KUKA KRL program: MyProgram_136().src

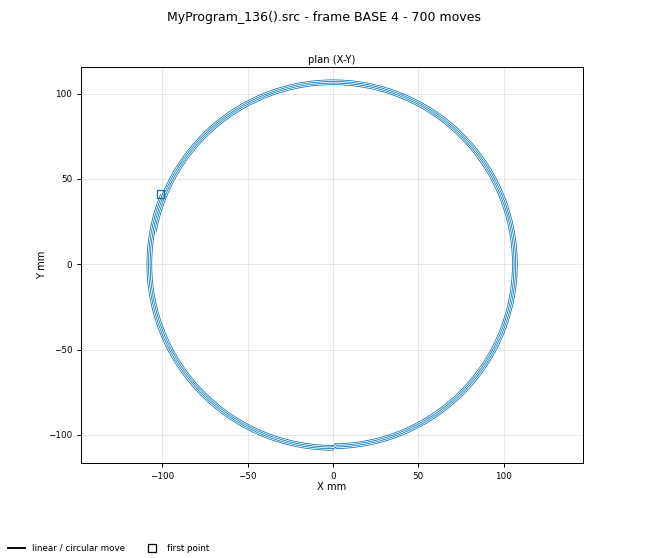
[picture p0: tool path of MyProgram_136().src in frame BASE 4, 700 of 700 moves have a stored position in this frame; points joined in program order, loops and branches not executed]
&ACCESS RVP
&REL 1
&PARAM TEMPLATE = C:\KRC\Roboter\Template\vorgabe
&PARAM EDITMASK = *
DEF MyProgram_136()
; ---- Setting reference (Base) ----
$BASE = BASE_DATA[4]

; --------------------------
; ---- Setting tool (TCP) ----
$TOOL = TOOL_DATA[3]
; --------------------------

$VEL.CP = VEL_APROX_PRINT
Startdeposition()
$VEL.CP = VEL_PRINT
LIN {X -101.0459,Y 40.9504,Z 110,A 153.8503,B 24.9356,C -1.8541,E1 24.8512,E2 291.8674} C_DIS
LIN {X -102.4048,Y 37.4224,Z 110,A 155.9368,B 24.9357,C -1.8516,E1 24.8492,E2 289.7749} C_DIS
LIN {X -103.4357,Y 34.473,Z 110,A 157.5676,B 24.9361,C -1.8461,E1 24.8477,E2 288.1481} C_DIS
LIN {X -104.6474,Y 30.5989,Z 110,A 159.7018,B 24.9366,C -1.8394,E1 24.846,E2 286.0176} C_DIS
LIN {X -105.5429,Y 27.3483,Z 110,A 161.5611,B 24.9367,C -1.837,E1 24.8446,E2 284.1531} C_DIS
LIN {X -106.3392,Y 24.0704,Z 110,A 163.3808,B 24.937,C -1.8331,E1 24.8435,E2 282.332} C_DIS
LIN {X -106.8901,Y 21.4916,Z 110,A 164.9562,B 24.9368,C -1.8358,E1 24.8426,E2 280.7408} C_DIS
LIN {X -107.8686,Y 15.8696,Z 110,A 167.7801,B 24.9379,C -1.8195,E1 24.8413,E2 277.9391} C_DIS
LIN {X -108.3438,Y 12.2078,Z 110,A 170.4812,B 24.9364,C -1.8421,E1 24.8404,E2 275.168} C_DIS
LIN {X -108.7748,Y 7.4321,Z 110,A 172.0604,B 24.9394,C -1.7983,E1 24.8401,E2 273.6837} C_DIS
LIN {X -109.0243,Y 1.0365,Z 110,A 175.4778,B 24.94,C -1.7893,E1 24.8398,E2 270.2672} C_DIS
LIN {X -108.9337,Y -4.5435,Z 110,A 179.2186,B 24.9386,C -1.8105,E1 24.8401,E2 266.4534} C_DIS
LIN {X -108.6738,Y -8.7861,Z 110,A -179.1678,B 24.9406,C -1.7797,E1 24.8404,E2 264.9035} C_DIS
LIN {X -108.4394,Y -11.3169,Z 110,A -177.6162,B 24.9404,C -1.7836,E1 24.8409,E2 263.3332} C_DIS
LIN {X -107.6634,Y -17.2072,Z 110,A -174.7453,B 24.9417,C -1.7642,E1 24.842,E2 260.4916} C_DIS
LIN {X -106.9005,Y -21.4409,Z 110,A -172.3194,B 24.9417,C -1.7633,E1 24.8432,E2 258.0534} C_DIS
LIN {X -106.0833,Y -25.1782,Z 110,A -170.3045,B 24.9421,C -1.7572,E1 24.8445,E2 256.0412} C_DIS
LIN {X -105.2578,Y -28.4248,Z 110,A -168.6511,B 24.9427,C -1.7478,E1 24.8456,E2 254.4007} C_DIS
LIN {X -104.3481,Y -31.6078,Z 110,A -166.7945,B 24.9428,C -1.7469,E1 24.8471,E2 252.5355} C_DIS
LIN {X -103.3127,Y -34.8378,Z 110,A -165.0254,B 24.9432,C -1.7411,E1 24.8487,E2 250.7702} C_DIS
LIN {X -102.0795,Y -38.3024,Z 110,A -163.1309,B 24.9437,C -1.7339,E1 24.8505,E2 248.8821} C_DIS
LIN {X -100.0319,Y -43.3688,Z 110,A -160.4375,B 24.9446,C -1.7187,E1 24.8533,E2 246.2098} C_DIS
LIN {X -98.1863,Y -47.399,Z 110,A -157.8891,B 24.9446,C -1.7204,E1 24.8563,E2 243.6435} C_DIS
LIN {X -96.4981,Y -50.7474,Z 110,A -155.8502,B 24.9447,C -1.7176,E1 24.8589,E2 241.6005} C_DIS
LIN {X -94.7103,Y -54.0117,Z 110,A -153.865,B 24.945,C -1.7134,E1 24.8616,E2 239.6149} C_DIS
LIN {X -91.6565,Y -59.0449,Z 110,A -150.4776,B 24.9448,C -1.7165,E1 24.8667,E2 236.2027} C_DIS
LIN {X -88.8476,Y -63.1926,Z 110,A -148.2791,B 24.9463,C -1.6931,E1 24.8701,E2 234.0492} C_DIS
LIN {X -86.6848,Y -66.1302,Z 110,A -146.1765,B 24.9461,C -1.6955,E1 24.8736,E2 231.9307} C_DIS
LIN {X -84.5749,Y -68.8062,Z 110,A -144.3868,B 24.9464,C -1.6912,E1 24.8768,E2 230.1428} C_DIS
LIN {X -82.6969,Y -71.0536,Z 110,A -142.3954,B 24.9455,C -1.7053,E1 24.8805,E2 228.1088} C_DIS
LIN {X -80.2724,Y -73.7802,Z 110,A -140.9176,B 24.9469,C -1.6838,E1 24.8832,E2 226.6757} C_DIS
LIN {X -77.6379,Y -76.5476,Z 110,A -139.1883,B 24.9478,C -1.6686,E1 24.8865,E2 224.9752} C_DIS
LIN {X -75.502,Y -78.6554,Z 110,A -137.3296,B 24.9473,C -1.6763,E1 24.8902,E2 223.0904} C_DIS
LIN {X -72.5889,Y -81.3515,Z 110,A -135.2119,B 24.9475,C -1.6733,E1 24.8946,E2 220.9713} C_DIS
LIN {X -69.8379,Y -83.725,Z 110,A -132.8251,B 24.9466,C -1.6885,E1 24.8998,E2 218.539} C_DIS
LIN {X -66.8378,Y -86.1396,Z 110,A -131.2769,B 24.948,C -1.666,E1 24.9031,E2 217.0388} C_DIS
LIN {X -63.7429,Y -88.455,Z 110,A -129.2893,B 24.9483,C -1.6607,E1 24.9076,E2 215.0566} C_DIS
LIN {X -60.5392,Y -90.6784,Z 110,A -127.116,B 24.9483,C -1.6623,E1 24.9126,E2 212.8724} C_DIS
LIN {X -55.2575,Y -93.9885,Z 110,A -123.6526,B 24.9481,C -1.6649,E1 24.9209,E2 209.392} C_DIS
LIN {X -51.1504,Y -96.2858,Z 110,A -121.304,B 24.9486,C -1.6566,E1 24.9266,E2 207.0566} C_DIS
LIN {X -46.668,Y -98.5376,Z 110,A -118.6742,B 24.9488,C -1.6531,E1 24.9332,E2 204.4282} C_DIS
LIN {X -43.398,Y -100.0191,Z 110,A -116.9327,B 24.9493,C -1.6452,E1 24.9376,E2 202.7013} C_DIS
LIN {X -39.7895,Y -101.5085,Z 110,A -114.827,B 24.9493,C -1.6453,E1 24.9431,E2 200.5906} C_DIS
LIN {X -36.1315,Y -102.8674,Z 110,A -112.8041,B 24.9495,C -1.6424,E1 24.9484,E2 198.5706} C_DIS
LIN {X -33.5707,Y -103.7313,Z 110,A -111.2544,B 24.9492,C -1.6465,E1 24.9525,E2 197.0083} C_DIS
LIN {X -28.2847,Y -105.2957,Z 110,A -108.424,B 24.9495,C -1.6418,E1 24.9601,E2 194.1844} C_DIS
LIN {X -25.199,Y -106.0784,Z 110,A -106.2515,B 24.9483,C -1.6615,E1 24.9662,E2 191.9624} C_DIS
LIN {X -21.329,Y -106.9234,Z 110,A -104.7514,B 24.9498,C -1.6366,E1 24.9701,E2 190.5195} C_DIS
LIN {X -17.6406,Y -107.5923,Z 110,A -102.8021,B 24.9499,C -1.6351,E1 24.9755,E2 188.5718} C_DIS
LIN {X -14.2432,Y -108.0942,Z 110,A -101.1009,B 24.9502,C -1.6305,E1 24.9801,E2 186.8803} C_DIS
LIN {X -11.5445,Y -108.4156,Z 110,A -99.5635,B 24.9499,C -1.6348,E1 24.9844,E2 185.3317} C_DIS
LIN {X -8.3441,Y -108.7091,Z 110,A -97.7326,B 24.9496,C -1.6406,E1 24.9896,E2 183.4862} C_DIS
LIN {X -4.4559,Y -108.9375,Z 110,A -95.6989,B 24.9496,C -1.6402,E1 24.9952,E2 181.4529} C_DIS
LIN {X -0.5852,Y -109.0268,Z 110,A -93.7792,B 24.9499,C -1.6358,E1 25.0006,E2 179.5435} C_DIS
LIN {X -0.5852,Y -109.0268,Z 110,A -93.7792,B 24.9499,C -1.6358,E1 25.0006,E2 179.5435} C_DIS
Enddeposition()
LIN {X 0.7508,Y -108.0795,Z 110,A -93.2455,B 24.9493,C -1.6454,E1 25.0021,E2 178.9871} C_DIS
Startdeposition()
$VEL.CP = VEL_PRINT
LIN {X -2.9231,Y -108.0454,Z 110,A -95.8982,B 24.9511,C -1.6161,E1 24.9945,E2 181.7093} C_DIS
LIN {X -6.8398,Y -107.8686,Z 110,A -97.972,B 24.9511,C -1.6161,E1 24.9888,E2 183.7836} C_DIS
LIN {X -10.1831,Y -107.6038,Z 110,A -99.6434,B 24.9508,C -1.6206,E1 24.9841,E2 185.4454} C_DIS
LIN {X -13.0586,Y -107.2936,Z 110,A -101.1347,B 24.9507,C -1.6224,E1 24.98,E2 186.9331} C_DIS
LIN {X -16.4613,Y -106.8234,Z 110,A -103.3915,B 24.9517,C -1.6054,E1 24.9737,E2 189.2322} C_DIS
LIN {X -19.6265,Y -106.2886,Z 110,A -104.6024,B 24.9505,C -1.6256,E1 24.9705,E2 190.3964} C_DIS
LIN {X -24.2676,Y -105.3247,Z 110,A -107.2289,B 24.9507,C -1.6222,E1 24.9633,E2 193.0342} C_DIS
LIN {X -30.7493,Y -103.618,Z 110,A -110.7194,B 24.9504,C -1.6269,E1 24.9539,E2 196.5189} C_DIS
LIN {X -33.1251,Y -102.8832,Z 110,A -112.13,B 24.9506,C -1.6242,E1 24.9501,E2 197.9384} C_DIS
LIN {X -36.5679,Y -101.7116,Z 110,A -114.1221,B 24.9506,C -1.6233,E1 24.9448,E2 199.9365} C_DIS
LIN {X -39.7247,Y -100.5197,Z 110,A -115.8285,B 24.9503,C -1.6283,E1 24.9404,E2 201.6347} C_DIS
LIN {X -42.6112,Y -99.3323,Z 110,A -117.5613,B 24.9504,C -1.6269,E1 24.9359,E2 203.3748} C_DIS
LIN {X -46.4464,Y -97.5966,Z 110,A -119.5451,B 24.9497,C -1.6392,E1 24.9309,E2 205.3343} C_DIS
LIN {X -48.7324,Y -96.476,Z 110,A -121.188,B 24.9503,C -1.6294,E1 24.9268,E2 207.0049} C_DIS
LIN {X -51.8131,Y -94.8562,Z 110,A -122.9938,B 24.95,C -1.6334,E1 24.9223,E2 208.8063} C_DIS
LIN {X -57.8107,Y -91.3266,Z 110,A -126.8101,B 24.95,C -1.6338,E1 24.9132,E2 212.6331} C_DIS
LIN {X -62.0089,Y -88.5283,Z 110,A -129.597,B 24.95,C -1.6339,E1 24.9067,E2 215.4292} C_DIS
LIN {X -64.932,Y -86.4062,Z 110,A -131.2208,B 24.9491,C -1.6484,E1 24.9031,E2 217.0242} C_DIS
LIN {X -70.239,Y -82.1506,Z 110,A -134.64,B 24.9482,C -1.6623,E1 24.8958,E2 220.4233} C_DIS
LIN {X -72.1623,Y -80.4663,Z 110,A -136.274,B 24.9487,C -1.6543,E1 24.8923,E2 222.0828} C_DIS
LIN {X -75.7805,Y -77.0687,Z 110,A -138.8814,B 24.9483,C -1.6606,E1 24.887,E2 224.6858} C_DIS
LIN {X -78.0174,Y -74.8036,Z 110,A -140.6814,B 24.9483,C -1.66,E1 24.8835,E2 226.4951} C_DIS
LIN {X -82.8135,Y -69.4577,Z 110,A -144.2462,B 24.9472,C -1.6778,E1 24.877,E2 230.0334} C_DIS
LIN {X -86.9571,Y -64.1939,Z 110,A -148.0447,B 24.9472,C -1.6771,E1 24.8704,E2 233.8517} C_DIS
LIN {X -89.1258,Y -61.1493,Z 110,A -150.2115,B 24.9474,C -1.6751,E1 24.8669,E2 236.0338} C_DIS
LIN {X -91.2432,Y -57.941,Z 110,A -152.5341,B 24.9477,C -1.6699,E1 24.8634,E2 238.3808} C_DIS
LIN {X -93.173,Y -54.782,Z 110,A -154.0573,B 24.9464,C -1.6914,E1 24.8613,E2 239.8604} C_DIS
LIN {X -95.078,Y -51.4044,Z 110,A -156.0328,B 24.9458,C -1.7,E1 24.8586,E2 241.8258} C_DIS
LIN {X -96.7287,Y -48.2268,Z 110,A -158.0219,B 24.9458,C -1.7019,E1 24.8561,E2 243.821} C_DIS
LIN {X -98.8506,Y -43.716,Z 110,A -160.6588,B 24.9452,C -1.7096,E1 24.853,E2 246.454} C_DIS
LIN {X -100.8213,Y -38.9567,Z 110,A -163.2646,B 24.9444,C -1.7222,E1 24.8503,E2 249.0443} C_DIS
LIN {X -102.0825,Y -35.517,Z 110,A -165.4232,B 24.9446,C -1.72,E1 24.8483,E2 251.2204} C_DIS
LIN {X -103.0681,Y -32.5499,Z 110,A -167.1107,B 24.9443,C -1.7239,E1 24.8468,E2 252.9084} C_DIS
LIN {X -104.0473,Y -29.2647,Z 110,A -168.7742,B 24.9436,C -1.7351,E1 24.8455,E2 254.5548} C_DIS
LIN {X -104.9195,Y -25.9661,Z 110,A -170.6629,B 24.9434,C -1.7377,E1 24.8442,E2 256.4482} C_DIS
LIN {X -105.7058,Y -22.5552,Z 110,A -172.6177,B 24.9433,C -1.7398,E1 24.843,E2 258.4095} C_DIS
LIN {X -106.6749,Y -17.4029,Z 110,A -175.1438,B 24.9421,C -1.7579,E1 24.8418,E2 260.9075} C_DIS
LIN {X -107.4911,Y -11.3081,Z 110,A -178.2308,B 24.941,C -1.7746,E1 24.8407,E2 263.9731} C_DIS
LIN {X -107.9447,Y -5.5101,Z 110,A 177.6041,B 24.9429,C -1.7449,E1 24.8399,E2 268.2341} C_DIS
LIN {X -108.0802,Y -1.0392,Z 110,A 176.1681,B 24.9402,C -1.7866,E1 24.8399,E2 269.5792} C_DIS
LIN {X -107.8861,Y 6.5706,Z 110,A 170.7512,B 24.9426,C -1.7495,E1 24.8404,E2 275.1172} C_DIS
LIN {X -107.3472,Y 12.601,Z 110,A 169.0253,B 24.9383,C -1.8138,E1 24.8409,E2 276.7001} C_DIS
LIN {X -106.5725,Y 18.0154,Z 110,A 165.5521,B 24.9391,C -1.8021,E1 24.8423,E2 280.222} C_DIS
LIN {X -105.91,Y 21.5708,Z 110,A 163.7053,B 24.9385,C -1.8108,E1 24.8433,E2 282.0589} C_DIS
LIN {X -105.0583,Y 25.3971,Z 110,A 161.6175,B 24.9381,C -1.8171,E1 24.8446,E2 284.1439} C_DIS
LIN {X -104.148,Y 28.9093,Z 110,A 159.1474,B 24.9391,C -1.8033,E1 24.8465,E2 286.6614} C_DIS
LIN {X -103.0003,Y 32.7633,Z 110,A 157.4686,B 24.9375,C -1.8264,E1 24.8478,E2 288.2945} C_DIS
LIN {X -101.7936,Y 36.3402,Z 110,A 155.2258,B 24.9376,C -1.8239,E1 24.8499,E2 290.5562} C_DIS
LIN {X -100.0581,Y 40.873,Z 110,A 152.9865,B 24.9363,C -1.844,E1 24.8522,E2 292.76} C_DIS
LIN {X -97.696,Y 46.2396,Z 110,A 149.9414,B 24.9354,C -1.8557,E1 24.8556,E2 295.7939} C_DIS
LIN {X -95.8219,Y 50.0053,Z 110,A 147.5969,B 24.9353,C -1.8581,E1 24.8586,E2 298.1452} C_DIS
LIN {X -94.2492,Y 52.909,Z 110,A 145.3421,B 24.9362,C -1.8448,E1 24.8617,E2 300.4437} C_DIS
LIN {X -92.3911,Y 56.0901,Z 110,A 143.8861,B 24.9345,C -1.8686,E1 24.8637,E2 301.8503} C_DIS
LIN {X -89.2594,Y 60.952,Z 110,A 140.8635,B 24.9338,C -1.8788,E1 24.8684,E2 304.8638} C_DIS
LIN {X -86.2572,Y 65.1305,Z 110,A 138.1262,B 24.9333,C -1.8859,E1 24.8728,E2 307.5976} C_DIS
LIN {X -83.4988,Y 68.6316,Z 110,A 135.6542,B 24.9332,C -1.8881,E1 24.8772,E2 310.0759} C_DIS
LIN {X -81.665,Y 70.8039,Z 110,A 133.7874,B 24.9338,C -1.8787,E1 24.8806,E2 311.9737} C_DIS
LIN {X -77.4056,Y 75.4383,Z 110,A 130.3591,B 24.9335,C -1.8836,E1 24.8872,E2 315.4051} C_DIS
LIN {X -75.0255,Y 77.8035,Z 110,A 129.4017,B 24.931,C -1.9185,E1 24.889,E2 316.2834} C_DIS
LIN {X -71.2242,Y 81.2979,Z 110,A 125.9153,B 24.9326,C -1.8968,E1 24.8963,E2 319.8355} C_DIS
LIN {X -66.9712,Y 84.8355,Z 110,A 123.3597,B 24.9311,C -1.9173,E1 24.9018,E2 322.3518} C_DIS
LIN {X -64.224,Y 86.935,Z 110,A 120.6363,B 24.9332,C -1.8879,E1 24.9081,E2 325.155} C_DIS
LIN {X -60.0312,Y 89.8826,Z 110,A 118.8337,B 24.9303,C -1.9275,E1 24.912,E2 326.8694} C_DIS
LIN {X -54.8633,Y 93.1249,Z 110,A 115.5325,B 24.9301,C -1.931,E1 24.9199,E2 330.1726} C_DIS
LIN {X -51.6981,Y 94.9187,Z 110,A 113.2966,B 24.9307,C -1.9227,E1 24.9254,E2 332.4348} C_DIS
LIN {X -44.9546,Y 98.2937,Z 110,A 109.657,B 24.9292,C -1.9427,E1 24.9344,E2 336.0363} C_DIS
LIN {X -38.6118,Y 100.9528,Z 110,A 105.8158,B 24.9294,C -1.9403,E1 24.9444,E2 339.8917} C_DIS
LIN {X -35.7699,Y 101.9937,Z 110,A 104.3216,B 24.929,C -1.9466,E1 24.9483,E2 341.3739} C_DIS
LIN {X -32.4367,Y 103.1032,Z 110,A 101.396,B 24.9317,C -1.9081,E1 24.9563,E2 344.3962} C_DIS
LIN {X -26.8495,Y 104.6963,Z 110,A 99.3346,B 24.9287,C -1.9503,E1 24.9616,E2 346.3605} C_DIS
LIN {X -22.3145,Y 105.7565,Z 110,A 96.6836,B 24.929,C -1.9454,E1 24.9689,E2 349.0264} C_DIS
LIN {X -18.9798,Y 106.4049,Z 110,A 94.4586,B 24.9301,C -1.9304,E1 24.9751,E2 351.2894} C_DIS
LIN {X -14.9308,Y 107.0484,Z 110,A 93.3607,B 24.927,C -1.9738,E1 24.9779,E2 352.2851} C_DIS
LIN {X -12.6887,Y 107.3369,Z 110,A 91.6804,B 24.9283,C -1.9555,E1 24.9826,E2 354.01} C_DIS
LIN {X -7.3361,Y 107.835,Z 110,A 89.198,B 24.9271,C -1.9714,E1 24.9894,E2 356.4559} C_DIS
LIN {X -2.7746,Y 108.05,Z 110,A 86.311,B 24.9284,C -1.9537,E1 24.9976,E2 359.3856} C_DIS
LIN {X 0.891,Y 108.0808,Z 110,A 84.4954,B 24.928,C -1.9591,E1 25.0026,E2 361.1882} C_DIS
LIN {X 5.9808,Y 107.9187,Z 110,A 81.4078,B 24.9292,C -1.9439,E1 25.0113,E2 364.311} C_DIS
LIN {X 11.3288,Y 107.4889,Z 110,A 78.9824,B 24.928,C -1.9603,E1 25.018,E2 366.6962} C_DIS
LIN {X 16.3757,Y 106.8366,Z 110,A 76.5404,B 24.9272,C -1.97,E1 25.0247,E2 369.1132} C_DIS
LIN {X 19.9462,Y 106.228,Z 110,A 74.3662,B 24.928,C -1.959,E1 25.0307,E2 371.3112} C_DIS
LIN {X 22.8813,Y 105.6347,Z 110,A 71.7891,B 24.931,C -1.9185,E1 25.038,E2 373.9807} C_DIS
LIN {X 28.1756,Y 104.3472,Z 110,A 69.8674,B 24.9283,C -1.9556,E1 25.0429,E2 375.8118} C_DIS
LIN {X 31.1953,Y 103.4857,Z 110,A 68.1558,B 24.9285,C -1.9524,E1 25.0475,E2 377.5278} C_DIS
LIN {X 34.636,Y 102.3844,Z 110,A 66.2894,B 24.9285,C -1.9529,E1 25.0525,E2 379.3897} C_DIS
LIN {X 38.0622,Y 101.1609,Z 110,A 64.3301,B 24.9287,C -1.9498,E1 25.0576,E2 381.3522} C_DIS
LIN {X 41.2095,Y 99.9211,Z 110,A 62.328,B 24.9295,C -1.9394,E1 25.0629,E2 383.3743} C_DIS
LIN {X 44.7362,Y 98.3921,Z 110,A 60.4093,B 24.9293,C -1.942,E1 25.0677,E2 385.2822} C_DIS
LIN {X 47.3331,Y 97.1705,Z 110,A 59.0667,B 24.9289,C -1.9474,E1 25.0711,E2 386.6083} C_DIS
LIN {X 50.2175,Y 95.7102,Z 110,A 56.4797,B 24.9317,C -1.9093,E1 25.0777,E2 389.2782} C_DIS
LIN {X 54.5861,Y 93.2888,Z 110,A 54.8061,B 24.929,C -1.9456,E1 25.0815,E2 390.8609} C_DIS
LIN {X 59.0506,Y 90.5291,Z 110,A 52.0056,B 24.9294,C -1.9406,E1 25.0882,E2 393.6645} C_DIS
LIN {X 61.8339,Y 88.6499,Z 110,A 50.1268,B 24.9299,C -1.9335,E1 25.0925,E2 395.5536} C_DIS
LIN {X 66.7509,Y 85.0096,Z 110,A 47.0934,B 24.9297,C -1.9365,E1 25.0993,E2 398.569} C_DIS
LIN {X 69.5993,Y 82.6956,Z 110,A 45.0071,B 24.9304,C -1.9269,E1 25.1038,E2 400.6702} C_DIS
LIN {X 72.9622,Y 79.7417,Z 110,A 42.5819,B 24.9309,C -1.9199,E1 25.1089,E2 403.1021} C_DIS
LIN {X 75.4849,Y 77.3607,Z 110,A 40.6308,B 24.9315,C -1.9113,E1 25.1128,E2 405.0655} C_DIS
LIN {X 79.5494,Y 73.1718,Z 110,A 37.8551,B 24.931,C -1.918,E1 25.1181,E2 407.8133} C_DIS
LIN {X 81.3856,Y 71.1237,Z 110,A 36.1979,B 24.9319,C -1.9062,E1 25.1212,E2 409.491} C_DIS
LIN {X 83.7596,Y 68.3129,Z 110,A 34.2472,B 24.9322,C -1.9016,E1 25.1247,E2 411.4437} C_DIS
LIN {X 85.7422,Y 65.8068,Z 110,A 32.5622,B 24.9325,C -1.8979,E1 25.1276,E2 413.1295} C_DIS
LIN {X 88.8564,Y 61.5368,Z 110,A 29.8153,B 24.9328,C -1.8932,E1 25.1321,E2 415.8741} C_DIS
LIN {X 91.094,Y 58.1735,Z 110,A 27.7873,B 24.9328,C -1.8925,E1 25.1352,E2 417.8937} C_DIS
LIN {X 92.4937,Y 55.9213,Z 110,A 26.2458,B 24.9335,C -1.8829,E1 25.1374,E2 419.45} C_DIS
LIN {X 94.9583,Y 51.6251,Z 110,A 23.6302,B 24.934,C -1.8762,E1 25.141,E2 422.0678} C_DIS
LIN {X 96.8679,Y 47.946,Z 110,A 21.0927,B 24.9355,C -1.8554,E1 25.1443,E2 424.6408} C_DIS
LIN {X 98.2909,Y 44.9609,Z 110,A 19.5229,B 24.9353,C -1.8583,E1 25.1461,E2 426.1954} C_DIS
LIN {X 100.0248,Y 40.9548,Z 110,A 17.407,B 24.9351,C -1.8601,E1 25.1484,E2 428.2953} C_DIS
LIN {X 101.3275,Y 37.6209,Z 110,A 15.4305,B 24.9358,C -1.8511,E1 25.1503,E2 430.2821} C_DIS
LIN {X 102.5279,Y 34.2104,Z 110,A 13.5485,B 24.9361,C -1.8468,E1 25.152,E2 432.1636} C_DIS
LIN {X 105.0686,Y 25.3549,Z 110,A 8.939,B 24.9363,C -1.8438,E1 25.1555,E2 436.7539} C_DIS
LIN {X 105.7303,Y 22.4405,Z 110,A 6.6665,B 24.9387,C -1.809,E1 25.1569,E2 439.0952} C_DIS
LIN {X 106.4713,Y 18.6104,Z 110,A 5.2526,B 24.9372,C -1.8308,E1 25.1576,E2 440.4493} C_DIS
LIN {X 107.1681,Y 14.0435,Z 110,A 2.7625,B 24.9378,C -1.8212,E1 25.1586,E2 442.9473} C_DIS
LIN {X 107.5322,Y 10.9152,Z 110,A 0.9649,B 24.9386,C -1.8103,E1 25.1591,E2 444.7601} C_DIS
LIN {X 107.9162,Y 6.0254,Z 110,A -1.8257,B 24.9397,C -1.7936,E1 25.1596,E2 447.5734} C_DIS
LIN {X 108.0691,Y 1.819,Z 110,A -3.6445,B 24.939,C -1.8044,E1 25.1598,E2 449.356} C_DIS
LIN {X 108.0751,Y -1.49,Z 110,A -5.9081,B 24.9408,C -1.7765,E1 25.1598,E2 451.672} C_DIS
LIN {X 107.9748,Y -4.8695,Z 110,A -6.8421,B 24.9387,C -1.8082,E1 25.1596,E2 452.5256} C_DIS
LIN {X 107.8463,Y -7.1695,Z 110,A -8.4766,B 24.9402,C -1.7861,E1 25.1594,E2 454.2026} C_DIS
LIN {X 107.5956,Y -10.2722,Z 110,A -10.1551,B 24.9407,C -1.7795,E1 25.1589,E2 455.8867} C_DIS
LIN {X 107.174,Y -13.9985,Z 110,A -12.0472,B 24.9408,C -1.7772,E1 25.1583,E2 457.7729} C_DIS
LIN {X 106.5691,Y -18.0356,Z 110,A -14.9658,B 24.9434,C -1.7374,E1 25.157,E2 460.7683} C_DIS
LIN {X 105.6802,Y -22.6722,Z 110,A -16.4996,B 24.9412,C -1.7715,E1 25.1562,E2 462.2128} C_DIS
LIN {X 103.8104,Y -30.1006,Z 110,A -20.6926,B 24.9424,C -1.7526,E1 25.1532,E2 466.426} C_DIS
LIN {X 102.8588,Y -33.2005,Z 110,A -23.1726,B 24.9449,C -1.7142,E1 25.151,E2 468.9827} C_DIS
LIN {X 101.3163,Y -37.6515,Z 110,A -24.907,B 24.9433,C -1.7394,E1 25.1495,E2 470.6478} C_DIS
LIN {X 100.2935,Y -40.2947,Z 110,A -26.504,B 24.9439,C -1.7306,E1 25.1478,E2 472.2567} C_DIS
LIN {X 98.9434,Y -43.5032,Z 110,A -28.5826,B 24.9449,C -1.7149,E1 25.1455,E2 474.3612} C_DIS
LIN {X 96.9914,Y -47.6969,Z 110,A -30.4686,B 24.9438,C -1.7321,E1 25.1433,E2 476.1963} C_DIS
LIN {X 94.7192,Y -52.0657,Z 110,A -33.2149,B 24.9447,C -1.7183,E1 25.1397,E2 478.9605} C_DIS
LIN {X 92.5424,Y -55.841,Z 110,A -35.8985,B 24.9461,C -1.6954,E1 25.1358,E2 481.6844} C_DIS
LIN {X 88.4528,Y -62.1175,Z 110,A -39.4593,B 24.9457,C -1.702,E1 25.1304,E2 485.212} C_DIS
LIN {X 85.7869,Y -65.7487,Z 110,A -42.011,B 24.9466,C -1.6884,E1 25.1261,E2 487.7836} C_DIS
LIN {X 84.1163,Y -67.8727,Z 110,A -44.1306,B 24.9487,C -1.6551,E1 25.1222,E2 489.972} C_DIS
LIN {X 80.8896,Y -71.6894,Z 110,A -45.8345,B 24.9466,C -1.6887,E1 25.1193,E2 491.5887} C_DIS
LIN {X 76.9703,Y -75.8801,Z 110,A -48.9773,B 24.9473,C -1.6767,E1 25.1132,E2 494.7462} C_DIS
LIN {X 72.6797,Y -80.001,Z 110,A -52.0202,B 24.9475,C -1.6739,E1 25.1071,E2 497.7832} C_DIS
LIN {X 70.6105,Y -81.8339,Z 110,A -54.0462,B 24.9492,C -1.6466,E1 25.1026,E2 499.8659} C_DIS
LIN {X 67.9897,Y -84.0215,Z 110,A -55.1935,B 24.9477,C -1.6708,E1 25.1003,E2 500.9514} C_DIS
LIN {X 64.577,Y -86.6729,Z 110,A -57.5918,B 24.9483,C -1.6613,E1 25.095,E2 503.3636} C_DIS
LIN {X 62.516,Y -88.1707,Z 110,A -59.9087,B 24.951,C -1.6176,E1 25.0895,E2 505.7757} C_DIS
LIN {X 58.0762,Y -91.1565,Z 110,A -62.1531,B 24.9498,C -1.6369,E1 25.0843,E2 507.9671} C_DIS
LIN {X 54.4372,Y -93.3768,Z 110,A -64.2061,B 24.9495,C -1.6414,E1 25.0794,E2 510.0031} C_DIS
LIN {X 48.2727,Y -96.706,Z 110,A -67.6459,B 24.9492,C -1.6466,E1 25.071,E2 513.4208} C_DIS
LIN {X 42.7542,Y -99.2699,Z 110,A -70.9102,B 24.9496,C -1.6399,E1 25.0627,E2 516.6928} C_DIS
LIN {X 40.1297,Y -100.3606,Z 110,A -72.6578,B 24.9504,C -1.6276,E1 25.0581,E2 518.4655} C_DIS
LIN {X 36.3792,Y -101.7799,Z 110,A -74.5355,B 24.9499,C -1.6352,E1 25.0532,E2 520.3214} C_DIS
LIN {X 32.2617,Y -103.1574,Z 110,A -77.7499,B 24.9524,C -1.5945,E1 25.0445,E2 523.626} C_DIS
LIN {X 27.3681,Y -104.563,Z 110,A -79.8519,B 24.9511,C -1.6163,E1 25.0389,E2 525.6732} C_DIS
LIN {X 23.5665,Y -105.4852,Z 110,A -81.7368,B 24.9507,C -1.6221,E1 25.0338,E2 527.5417} C_DIS
LIN {X 20.2277,Y -106.1748,Z 110,A -84.7357,B 24.9537,C -1.5719,E1 25.0253,E2 530.656} C_DIS
LIN {X 13.5039,Y -107.2381,Z 110,A -86.7579,B 24.95,C -1.6342,E1 25.0201,E2 532.529} C_DIS
LIN {X 9.385,Y -107.6774,Z 110,A -89.3817,B 24.9511,C -1.6153,E1 25.0127,E2 535.1958} C_DIS
LIN {X 5.6705,Y -107.9358,Z 110,A -91.2473,B 24.9509,C -1.6189,E1 25.0075,E2 537.0521} C_DIS
LIN {X 2.0664,Y -108.0645,Z 110,A -93.1794,B 24.9509,C -1.6175,E1 25.0021,E2 538.9871} C_DIS
LIN {X 2.0664,Y -108.0645,Z 110,A -93.1794,B 24.9509,C -1.6175,E1 25.0021,E2 538.9871} C_DIS
Enddeposition()
LIN {X 0.7521,Y -107.1372,Z 110,A -93.9447,B 24.9501,C -1.6312,E1 25.0001,E2 539.72} C_DIS
Startdeposition()
$VEL.CP = VEL_PRINT
LIN {X 4.4852,Y -107.0463,Z 110,A -91.0973,B 24.948,C -1.6664,E1 25.0083,E2 536.7897} C_DIS
LIN {X 8.1816,Y -106.8279,Z 110,A -89.0915,B 24.9478,C -1.6683,E1 25.0139,E2 534.7801} C_DIS
LIN {X 11.6155,Y -106.5097,Z 110,A -87.2836,B 24.9478,C -1.6678,E1 25.0189,E2 532.9746} C_DIS
LIN {X 17.6369,Y -105.6786,Z 110,A -83.4506,B 24.9462,C -1.6944,E1 25.0296,E2 529.0822} C_DIS
LIN {X 21.6328,Y -104.9335,Z 110,A -82.0133,B 24.948,C -1.6655,E1 25.0334,E2 527.7151} C_DIS
LIN {X 27.0894,Y -103.6599,Z 110,A -78.6291,B 24.9468,C -1.6846,E1 25.0427,E2 524.2906} C_DIS
LIN {X 31.9007,Y -102.281,Z 110,A -76.3045,B 24.9476,C -1.6729,E1 25.0488,E2 521.9977} C_DIS
LIN {X 34.7005,Y -101.3663,Z 110,A -74.5285,B 24.9469,C -1.6833,E1 25.0536,E2 520.2005} C_DIS
LIN {X 38.5831,Y -99.9531,Z 110,A -72.4211,B 24.9469,C -1.682,E1 25.059,E2 518.1008} C_DIS
LIN {X 41.7204,Y -98.6835,Z 110,A -70.3475,B 24.9461,C -1.6958,E1 25.0645,E2 515.9993} C_DIS
LIN {X 48.2086,Y -95.6835,Z 110,A -66.9197,B 24.9468,C -1.6851,E1 25.073,E2 512.6057} C_DIS
LIN {X 52.1087,Y -93.6148,Z 110,A -64.7961,B 24.9472,C -1.6791,E1 25.0782,E2 510.5022} C_DIS
LIN {X 55.5143,Y -91.6363,Z 110,A -62.2296,B 24.9457,C -1.7026,E1 25.0845,E2 507.8881} C_DIS
LIN {X 60.4854,Y -88.4345,Z 110,A -59.1691,B 24.9456,C -1.7045,E1 25.0916,E2 504.8333} C_DIS
LIN {X 63.3708,Y -86.3896,Z 110,A -57.3633,B 24.9456,C -1.7047,E1 25.0957,E2 503.0333} C_DIS
LIN {X 67.4191,Y -83.2687,Z 110,A -53.729,B 24.9426,C -1.7498,E1 25.1038,E2 499.3061} C_DIS
LIN {X 71.4582,Y -79.8295,Z 110,A -52.0456,B 24.9454,C -1.7063,E1 25.1072,E2 497.7321} C_DIS
LIN {X 75.7315,Y -75.7901,Z 110,A -48.1605,B 24.9429,C -1.7459,E1 25.1151,E2 493.7697} C_DIS
LIN {X 78.2593,Y -73.1749,Z 110,A -46.5337,B 24.9435,C -1.7369,E1 25.1182,E2 492.1711} C_DIS
LIN {X 82.1599,Y -68.7671,Z 110,A -43.315,B 24.9427,C -1.7482,E1 25.124,E2 488.9404} C_DIS
LIN {X 86.1549,Y -63.6914,Z 110,A -40.3246,B 24.9434,C -1.7373,E1 25.1291,E2 485.9898} C_DIS
LIN {X 87.8401,Y -61.3448,Z 110,A -38.639,B 24.9428,C -1.7477,E1 25.1318,E2 484.2879} C_DIS
LIN {X 90.3252,Y -57.6235,Z 110,A -36.296,B 24.9425,C -1.7523,E1 25.1354,E2 481.9457} C_DIS
LIN {X 92.2638,Y -54.4648,Z 110,A -34.209,B 24.9418,C -1.7626,E1 25.1384,E2 479.845} C_DIS
LIN {X 93.9085,Y -51.5803,Z 110,A -32.1707,B 24.9407,C -1.7793,E1 25.1412,E2 477.7779} C_DIS
LIN {X 95.5759,Y -48.4191,Z 110,A -30.5854,B 24.9412,C -1.7707,E1 25.1432,E2 476.2214} C_DIS
LIN {X 98.0663,Y -43.1527,Z 110,A -27.7419,B 24.9414,C -1.7683,E1 25.1466,E2 473.399} C_DIS
LIN {X 98.9006,Y -41.2054,Z 110,A -26.0889,B 24.9396,C -1.7946,E1 25.1484,E2 471.6931} C_DIS
LIN {X 100.5073,Y -37.1145,Z 110,A -23.393,B 24.9381,C -1.8172,E1 25.1511,E2 468.959} C_DIS
LIN {X 101.9342,Y -32.9916,Z 110,A -22.1378,B 24.9408,C -1.777,E1 25.1521,E2 467.8055} C_DIS
LIN {X 103.116,Y -29.0882,Z 110,A -18.706,B 24.9366,C -1.8391,E1 25.1549,E2 464.2469} C_DIS
LIN {X 104.4158,Y -24.008,Z 110,A -16.8514,B 24.9389,C -1.806,E1 25.156,E2 462.4811} C_DIS
LIN {X 105.1274,Y -20.6743,Z 110,A -14.64,B 24.9373,C -1.829,E1 25.1572,E2 460.2284} C_DIS
LIN {X 106.1698,Y -14.3986,Z 110,A -11.5101,B 24.9373,C -1.828,E1 25.1585,E2 457.1193} C_DIS
LIN {X 106.5881,Y -10.8669,Z 110,A -9.6024,B 24.9369,C -1.8344,E1 25.1591,E2 455.2076} C_DIS
LIN {X 106.9056,Y -7.0871,Z 110,A -7.6765,B 24.9368,C -1.8365,E1 25.1595,E2 453.2883} C_DIS
LIN {X 107.139,Y -0.6133,Z 110,A -4.5698,B 24.9371,C -1.832,E1 25.1598,E2 450.2107} C_DIS
LIN {X 107.1219,Y 1.9787,Z 110,A -2.2831,B 24.934,C -1.8761,E1 25.1597,E2 447.8335} C_DIS
LIN {X 106.9663,Y 6.1045,Z 110,A -0.1528,B 24.9338,C -1.8798,E1 25.1593,E2 445.7073} C_DIS
LIN {X 106.6774,Y 9.9485,Z 110,A 1.2618,B 24.9353,C -1.8579,E1 25.159,E2 444.3526} C_DIS
LIN {X 106.3413,Y 13.0742,Z 110,A 3.845,B 24.9321,C -1.903,E1 25.1581,E2 441.6783} C_DIS
LIN {X 105.62,Y 17.987,Z 110,A 5.5132,B 24.9346,C -1.868,E1 25.1574,E2 440.1026} C_DIS
LIN {X 104.6324,Y 23.0463,Z 110,A 8.1747,B 24.9343,C -1.8724,E1 25.156,E2 437.4461} C_DIS
LIN {X 104.0712,Y 25.4598,Z 110,A 9.6909,B 24.9334,C -1.8849,E1 25.1549,E2 435.9094} C_DIS
LIN {X 102.1738,Y 32.2462,Z 110,A 13.5736,B 24.9322,C -1.9013,E1 25.1519,E2 432.0101} C_DIS
LIN {X 101.0153,Y 35.7071,Z 110,A 15.3668,B 24.9323,C -1.9002,E1 25.1503,E2 430.2295} C_DIS
LIN {X 99.7734,Y 39.0423,Z 110,A 17.2677,B 24.9319,C -1.9058,E1 25.1484,E2 428.3261} C_DIS
LIN {X 98.5508,Y 42.0354,Z 110,A 19.0726,B 24.9313,C -1.9141,E1 25.1465,E2 426.5116} C_DIS
LIN {X 97.4877,Y 44.4454,Z 110,A 20.4683,B 24.9311,C -1.9175,E1 25.1448,E2 425.1153} C_DIS
LIN {X 95.347,Y 48.867,Z 110,A 22.92,B 24.9311,C -1.9173,E1 25.1418,E2 422.6772} C_DIS
LIN {X 93.8573,Y 51.6739,Z 110,A 24.9238,B 24.9298,C -1.9352,E1 25.1391,E2 420.6418} C_DIS
LIN {X 91.4358,Y 55.8441,Z 110,A 27.2476,B 24.9301,C -1.9311,E1 25.1358,E2 418.3395} C_DIS
LIN {X 88.9977,Y 59.6546,Z 110,A 29.6298,B 24.9297,C -1.9358,E1 25.1322,E2 415.9582} C_DIS
LIN {X 86.3602,Y 63.4111,Z 110,A 32.0243,B 24.9295,C -1.9394,E1 25.1284,E2 413.5669} C_DIS
LIN {X 84.6907,Y 65.6247,Z 110,A 33.6752,B 24.9287,C -1.9502,E1 25.1255,E2 411.8983} C_DIS
LIN {X 82.3558,Y 68.5313,Z 110,A 35.568,B 24.9287,C -1.9506,E1 25.1222,E2 410.0132} C_DIS
LIN {X 79.9649,Y 71.3069,Z 110,A 37.8385,B 24.9274,C -1.9684,E1 25.1179,E2 407.7107} C_DIS
LIN {X 76.1931,Y 75.3236,Z 110,A 40.0459,B 24.9292,C -1.9435,E1 25.1138,E2 405.5719} C_DIS
LIN {X 74.4049,Y 77.0905,Z 110,A 41.8041,B 24.9277,C -1.9638,E1 25.1102,E2 403.7729} C_DIS
LIN {X 71.7283,Y 79.5877,Z 110,A 43.8333,B 24.9272,C -1.9709,E1 25.106,E2 401.7354} C_DIS
LIN {X 69.1063,Y 81.8754,Z 110,A 45.7534,B 24.9267,C -1.977,E1 25.1019,E2 399.8083} C_DIS
LIN {X 64.9961,Y 85.173,Z 110,A 48.7014,B 24.9259,C -1.9877,E1 25.0954,E2 396.846} C_DIS
LIN {X 60.9805,Y 88.0934,Z 110,A 51.099,B 24.9264,C -1.9813,E1 25.09,E2 394.4717} C_DIS
LIN {X 58.4745,Y 89.7781,Z 110,A 52.9122,B 24.9256,C -1.9922,E1 25.0857,E2 392.6386} C_DIS
LIN {X 55.5529,Y 91.6128,Z 110,A 54.5302,B 24.9261,C -1.9856,E1 25.0819,E2 391.0416} C_DIS
LIN {X 50.6435,Y 94.4167,Z 110,A 57.4488,B 24.9261,C -1.9854,E1 25.0749,E2 388.1319} C_DIS
LIN {X 47.7127,Y 95.9299,Z 110,A 59.2542,B 24.9258,C -1.9894,E1 25.0703,E2 386.322} C_DIS
LIN {X 44.6549,Y 97.3921,Z 110,A 60.9523,B 24.926,C -1.9869,E1 25.0661,E2 384.6343} C_DIS
LIN {X 40.7385,Y 99.0936,Z 110,A 63.3731,B 24.9254,C -1.995,E1 25.0598,E2 382.2} C_DIS
LIN {X 37.5994,Y 100.3267,Z 110,A 65.2525,B 24.925,C -1.9999,E1 25.0549,E2 380.3131} C_DIS
LIN {X 34.2435,Y 101.5204,Z 110,A 67.0453,B 24.9252,C -1.997,E1 25.0502,E2 378.5308} C_DIS
LIN {X 30.7669,Y 102.628,Z 110,A 69.0527,B 24.9249,C -2.0007,E1 25.0448,E2 376.5181} C_DIS
LIN {X 27.6284,Y 103.5171,Z 110,A 71.385,B 24.923,C -2.026,E1 25.0384,E2 374.1296} C_DIS
LIN {X 23.4668,Y 104.5406,Z 110,A 72.9537,B 24.9252,C -1.9976,E1 25.0343,E2 372.6303} C_DIS
LIN {X 19.5983,Y 105.3341,Z 110,A 75.6229,B 24.9234,C -2.0212,E1 25.0269,E2 369.9084} C_DIS
LIN {X 16.1863,Y 105.9106,Z 110,A 77.7427,B 24.9225,C -2.0327,E1 25.0209,E2 367.7632} C_DIS
LIN {X 11.5399,Y 106.5176,Z 110,A 79.299,B 24.9254,C -1.9947,E1 25.0169,E2 366.2982} C_DIS
LIN {X 5.2493,Y 107.0124,Z 110,A 83.6079,B 24.9225,C -2.0324,E1 25.0046,E2 361.9018} C_DIS
LIN {X 0.6954,Y 107.1379,Z 110,A 84.9405,B 24.9259,C -1.9878,E1 25.0012,E2 360.6751} C_DIS
LIN {X -1.7907,Y 107.1254,Z 110,A 87.5529,B 24.9221,C -2.0388,E1 24.9936,E2 357.9417} C_DIS
LIN {X -7.1078,Y 106.9042,Z 110,A 89.1582,B 24.9259,C -1.9882,E1 24.9894,E2 356.4559} C_DIS
LIN {X -12.5475,Y 106.4029,Z 110,A 92.4275,B 24.925,C -2.0004,E1 24.9803,E2 353.1559} C_DIS
LIN {X -18.7539,Y 105.4863,Z 110,A 95.7447,B 24.9253,C -1.9965,E1 24.9711,E2 349.845} C_DIS
LIN {X -24.4074,Y 104.3235,Z 110,A 98.7526,B 24.9257,C -1.9907,E1 24.9629,E2 346.8472} C_DIS
LIN {X -26.994,Y 103.6844,Z 110,A 100.2957,B 24.9255,C -1.9939,E1 24.9587,E2 345.2943} C_DIS
LIN {X -32.6278,Y 102.0519,Z 110,A 103.29,B 24.9261,C -1.9849,E1 24.9508,E2 342.3165} C_DIS
LIN {X -35.4071,Y 101.1205,Z 110,A 105.0217,B 24.9258,C -1.9893,E1 24.9461,E2 340.571} C_DIS
LIN {X -41.8475,Y 98.63,Z 110,A 108.8044,B 24.9259,C -1.9877,E1 24.9363,E2 336.7839} C_DIS
LIN {X -45.2009,Y 97.1386,Z 110,A 110.6836,B 24.9264,C -1.9815,E1 24.9316,E2 334.9149} C_DIS
LIN {X -48.6276,Y 95.4693,Z 110,A 113.2189,B 24.9252,C -1.9973,E1 24.9251,E2 332.3352} C_DIS
LIN {X -51.8355,Y 93.7673,Z 110,A 114.516,B 24.9273,C -1.9692,E1 24.9221,E2 331.1013} C_DIS
LIN {X -57.8155,Y 90.202,Z 110,A 118.0637,B 24.9283,C -1.9557,E1 24.9137,E2 327.5749} C_DIS
LIN {X -63.3802,Y 86.3827,Z 110,A 121.6222,B 24.929,C -1.9465,E1 24.9055,E2 324.0262} C_DIS
LIN {X -65.3347,Y 84.9141,Z 110,A 123.3784,B 24.9279,C -1.9606,E1 24.9015,E2 322.23} C_DIS
LIN {X -68.2435,Y 82.595,Z 110,A 125.3799,B 24.9282,C -1.9567,E1 24.8971,E2 320.2302} C_DIS
LIN {X -72.5181,Y 78.8679,Z 110,A 128.4412,B 24.9287,C -1.9508,E1 24.8908,E2 317.1709} C_DIS
LIN {X -75.2858,Y 76.2304,Z 110,A 130.5255,B 24.9289,C -1.9474,E1 24.8866,E2 315.086} C_DIS
LIN {X -78.0496,Y 73.3981,Z 110,A 133.1717,B 24.9278,C -1.9621,E1 24.8814,E2 312.3933} C_DIS
LIN {X -80.7099,Y 70.4623,Z 110,A 134.7507,B 24.9297,C -1.9364,E1 24.8786,E2 310.8685} C_DIS
LIN {X -83.7745,Y 66.7909,Z 110,A 137.1327,B 24.9307,C -1.9231,E1 24.8744,E2 308.507} C_DIS
LIN {X -85.7122,Y 64.2841,Z 110,A 139.4255,B 24.9294,C -1.9409,E1 24.8704,E2 306.161} C_DIS
LIN {X -87.708,Y 61.5349,Z 110,A 140.7638,B 24.931,C -1.918,E1 24.8684,E2 304.8706} C_DIS
LIN {X -90.1207,Y 57.942,Z 110,A 142.8321,B 24.9322,C -1.9024,E1 24.8652,E2 302.8291} C_DIS
LIN {X -91.5303,Y 55.6887,Z 110,A 144.7583,B 24.9311,C -1.9171,E1 24.8623,E2 300.8582} C_DIS
LIN {X -93.68,Y 51.9918,Z 110,A 146.8449,B 24.9321,C -1.903,E1 24.8595,E2 298.7944} C_DIS
LIN {X -95.6641,Y 48.2441,Z 110,A 149.5016,B 24.9316,C -1.9107,E1 24.856,E2 296.1051} C_DIS
LIN {X -98.3767,Y 42.4407,Z 110,A 152.7361,B 24.9328,C -1.8931,E1 24.8523,E2 292.8946} C_DIS
LIN {X -99.8136,Y 38.9402,Z 110,A 154.6258,B 24.9336,C -1.882,E1 24.8504,E2 291.021} C_DIS
LIN {X -101.2582,Y 35.0146,Z 110,A 156.7747,B 24.9343,C -1.8718,E1 24.8484,E2 288.8843} C_DIS
LIN {X -102.0336,Y 32.6842,Z 110,A 158.5271,B 24.9335,C -1.8839,E1 24.8468,E2 287.0929} C_DIS
LIN {X -103.3996,Y 28.0634,Z 110,A 160.8463,B 24.9347,C -1.8662,E1 24.8451,E2 284.8025} C_DIS
LIN {X -104.3018,Y 24.5013,Z 110,A 162.8605,B 24.935,C -1.8617,E1 24.8437,E2 282.7872} C_DIS
LIN {X -105.0461,Y 21.0847,Z 110,A 164.8043,B 24.9353,C -1.8584,E1 24.8426,E2 280.8398} C_DIS
LIN {X -106.1607,Y 14.4671,Z 110,A 168.2899,B 24.9363,C -1.843,E1 24.8411,E2 277.3703} C_DIS
LIN {X -106.5717,Y 11.0233,Z 110,A 170.7514,B 24.9352,C -1.8595,E1 24.8404,E2 274.8547} C_DIS
LIN {X -106.9067,Y 7.071,Z 110,A 172.2646,B 24.9372,C -1.8301,E1 24.8401,E2 273.4025} C_DIS
LIN {X -107.1242,Y 1.8538,Z 110,A 175.0503,B 24.9379,C -1.8208,E1 24.8398,E2 270.6222} C_DIS
LIN {X -107.1363,Y -1.013,Z 110,A 176.7631,B 24.9377,C -1.8224,E1 24.8398,E2 268.8952} C_DIS
LIN {X -106.9584,Y -6.2474,Z 110,A 179.8955,B 24.9375,C -1.8257,E1 24.8402,E2 265.7361} C_DIS
LIN {X -106.7174,Y -9.5146,Z 110,A -178.7959,B 24.939,C -1.8036,E1 24.8405,E2 264.4723} C_DIS
LIN {X -106.3946,Y -12.619,Z 110,A -176.5274,B 24.9379,C -1.8206,E1 24.8413,E2 262.1498} C_DIS
LIN {X -105.8789,Y -16.3912,Z 110,A -175.2091,B 24.9401,C -1.7875,E1 24.8418,E2 260.9025} C_DIS
LIN {X -105.3419,Y -19.5566,Z 110,A -173.2526,B 24.9399,C -1.7909,E1 24.8427,E2 258.9263} C_DIS
LIN {X -104.6696,Y -22.8756,Z 110,A -171.4477,B 24.9403,C -1.785,E1 24.8438,E2 257.1248} C_DIS
LIN {X -103.7942,Y -26.5668,Z 110,A -169.4341,B 24.9407,C -1.7782,E1 24.8451,E2 255.1156} C_DIS
LIN {X -102.9041,Y -29.8352,Z 110,A -167.462,B 24.9407,C -1.7786,E1 24.8466,E2 253.1312} C_DIS
LIN {X -101.8002,Y -33.4057,Z 110,A -165.565,B 24.9414,C -1.7688,E1 24.8482,E2 251.2466} C_DIS
LIN {X -100.8397,Y -36.2031,Z 110,A -163.9133,B 24.9414,C -1.7667,E1 24.8498,E2 249.5906} C_DIS
LIN {X -99.3256,Y -40.1685,Z 110,A -161.3214,B 24.9411,C -1.7721,E1 24.8525,E2 246.9712} C_DIS
LIN {X -98.0737,Y -43.1356,Z 110,A -160.244,B 24.9431,C -1.7431,E1 24.8536,E2 245.9572} C_DIS
LIN {X -96.8417,Y -45.8378,Z 110,A -158.469,B 24.9429,C -1.7455,E1 24.8557,E2 244.1668} C_DIS
LIN {X -95.0602,Y -49.4256,Z 110,A -156.1231,B 24.9428,C -1.7471,E1 24.8587,E2 241.8043} C_DIS
LIN {X -93.3956,Y -52.5012,Z 110,A -154.3246,B 24.9433,C -1.7394,E1 24.8611,E2 240.0149} C_DIS
LIN {X -91.2726,Y -56.1127,Z 110,A -152.2157,B 24.944,C -1.7284,E1 24.8641,E2 237.9212} C_DIS
LIN {X -88.7219,Y -60.062,Z 110,A -149.6547,B 24.9443,C -1.7237,E1 24.868,E2 235.3585} C_DIS
LIN {X -87.0314,Y -62.4872,Z 110,A -147.8762,B 24.9441,C -1.7272,E1 24.8709,E2 233.563} C_DIS
LIN {X -82.8689,Y -67.9112,Z 110,A -144.5941,B 24.9456,C -1.7041,E1 24.8765,E2 230.3203} C_DIS
LIN {X -78.7019,Y -72.6991,Z 110,A -141.4544,B 24.9467,C -1.6866,E1 24.8822,E2 227.2081} C_DIS
LIN {X -76.0809,Y -75.4371,Z 110,A -138.83,B 24.9455,C -1.7049,E1 24.8873,E2 224.5288} C_DIS
LIN {X -72.275,Y -79.0911,Z 110,A -136.0743,B 24.9461,C -1.6965,E1 24.8929,E2 221.7817} C_DIS
LIN {X -69.6909,Y -81.3767,Z 110,A -133.2187,B 24.9438,C -1.7322,E1 24.8992,E2 218.8301} C_DIS
LIN {X -65.4506,Y -84.8248,Z 110,A -131.5872,B 24.9473,C -1.6767,E1 24.9025,E2 217.3247} C_DIS
LIN {X -61.676,Y -87.6099,Z 110,A -128.7905,B 24.9469,C -1.6834,E1 24.9088,E2 214.5022} C_DIS
LIN {X -58.8364,Y -89.5395,Z 110,A -126.8179,B 24.9467,C -1.6858,E1 24.9134,E2 212.5174} C_DIS
LIN {X -54.1718,Y -92.437,Z 110,A -124.0817,B 24.9475,C -1.6735,E1 24.9199,E2 209.8018} C_DIS
LIN {X -52.15,Y -93.5917,Z 110,A -122.6619,B 24.9472,C -1.6786,E1 24.9234,E2 208.3657} C_DIS
LIN {X -48.93,Y -95.3148,Z 110,A -120.5775,B 24.947,C -1.6813,E1 24.9286,E2 206.2693} C_DIS
LIN {X -45.5831,Y -96.9607,Z 110,A -118.5295,B 24.947,C -1.681,E1 24.9338,E2 204.2168} C_DIS
LIN {X -41.0015,Y -98.9865,Z 110,A -116.1027,B 24.9479,C -1.6681,E1 24.9399,E2 201.8149} C_DIS
LIN {X -37.568,Y -100.3386,Z 110,A -113.9353,B 24.9475,C -1.674,E1 24.9456,E2 199.629} C_DIS
LIN {X -34.1419,Y -101.5547,Z 110,A -112.1114,B 24.9479,C -1.6675,E1 24.9504,E2 197.8168} C_DIS
LIN {X -30.7856,Y -102.6225,Z 110,A -109.5208,B 24.9462,C -1.6946,E1 24.9575,E2 195.1577} C_DIS
LIN {X -26.5142,Y -103.8077,Z 110,A -107.9286,B 24.9483,C -1.6618,E1 24.9616,E2 193.6409} C_DIS
LIN {X -23.5713,Y -104.5166,Z 110,A -105.924,B 24.9473,C -1.6765,E1 24.9672,E2 191.5988} C_DIS
LIN {X -19.6722,Y -105.3204,Z 110,A -103.4088,B 24.9464,C -1.6913,E1 24.9742,E2 189.0456} C_DIS
LIN {X -15.3904,Y -106.0295,Z 110,A -102.0013,B 24.9488,C -1.6537,E1 24.9778,E2 187.7262} C_DIS
LIN {X -11.3585,Y -106.5366,Z 110,A -99.6355,B 24.9483,C -1.6611,E1 24.9844,E2 185.3412} C_DIS
LIN {X -8.2111,Y -106.8256,Z 110,A -97.8225,B 24.948,C -1.666,E1 24.9895,E2 183.5157} C_DIS
LIN {X -4.5534,Y -107.0434,Z 110,A -95.9886,B 24.9483,C -1.6611,E1 24.9946,E2 181.6932} C_DIS
LIN {X -1.2861,Y -107.1343,Z 110,A -94.036,B 24.9478,C -1.6697,E1 25.0001,E2 179.72} C_DIS
LIN {X -1.2861,Y -107.1343,Z 110,A -94.036,B 24.9478,C -1.6697,E1 25.0001,E2 179.72} C_DIS
Enddeposition()
LIN {X 0.7525,Y -106.1913,Z 110,A -93.9214,B 24.9492,C -1.647,E1 25.0003,E2 179.6592} C_DIS
Startdeposition()
$VEL.CP = VEL_PRINT
LIN {X -3.1055,Y -106.1508,Z 110,A -96.0482,B 24.9493,C -1.6448,E1 24.9943,E2 181.7914} C_DIS
LIN {X -6.5249,Y -105.9974,Z 110,A -97.9412,B 24.9494,C -1.6428,E1 24.989,E2 183.6896} C_DIS
LIN {X -10.4092,Y -105.6867,Z 110,A -100.173,B 24.9497,C -1.6378,E1 24.9828,E2 185.9343} C_DIS
LIN {X -14.1261,Y -105.2535,Z 110,A -102.4214,B 24.9503,C -1.6292,E1 24.9765,E2 188.2047} C_DIS
LIN {X -17.4311,Y -104.7558,Z 110,A -103.7714,B 24.9491,C -1.6475,E1 24.9729,E2 189.5126} C_DIS
LIN {X -21.2061,Y -104.0574,Z 110,A -105.8856,B 24.9491,C -1.6466,E1 24.9671,E2 191.6312} C_DIS
LIN {X -24.7246,Y -103.2789,Z 110,A -107.8934,B 24.9493,C -1.6451,E1 24.9616,E2 193.6453} C_DIS
LIN {X -29.5201,Y -102.0124,Z 110,A -110.441,B 24.9489,C -1.6518,E1 24.9548,E2 196.181} C_DIS
LIN {X -32.6174,Y -101.063,Z 110,A -112.2266,B 24.9489,C -1.6516,E1 24.95,E2 197.97} C_DIS
LIN {X -35.8298,Y -99.971,Z 110,A -114.1357,B 24.9489,C -1.6501,E1 24.9449,E2 199.8864} C_DIS
LIN {X -38.8678,Y -98.8277,Z 110,A -115.7741,B 24.9486,C -1.6562,E1 24.9407,E2 201.514} C_DIS
LIN {X -41.9693,Y -97.5523,Z 110,A -118.0027,B 24.9495,C -1.642,E1 24.9349,E2 203.7814} C_DIS
LIN {X -46.1448,Y -95.6467,Z 110,A -120.1148,B 24.9484,C -1.6588,E1 24.9296,E2 205.8589} C_DIS
LIN {X -49.2721,Y -94.0741,Z 110,A -121.969,B 24.9482,C -1.6625,E1 24.925,E2 207.7092} C_DIS
LIN {X -52.013,Y -92.5869,Z 110,A -123.8114,B 24.9484,C -1.6587,E1 24.9205,E2 209.566} C_DIS
LIN {X -54.6846,Y -91.0358,Z 110,A -125.5585,B 24.9484,C -1.6581,E1 24.9163,E2 211.3199} C_DIS
LIN {X -57.9266,Y -89.0086,Z 110,A -127.5012,B 24.948,C -1.6658,E1 24.9117,E2 213.2504} C_DIS
LIN {X -60.817,Y -87.0573,Z 110,A -129.4457,B 24.948,C -1.6665,E1 24.9072,E2 215.1998} C_DIS
LIN {X -63.9637,Y -84.7721,Z 110,A -131.2661,B 24.9471,C -1.6807,E1 24.9032,E2 216.993} C_DIS
LIN {X -68.5376,Y -81.1197,Z 110,A -134.6613,B 24.9473,C -1.6776,E1 24.8958,E2 220.4083} C_DIS
LIN {X -71.4597,Y -78.5578,Z 110,A -137.0088,B 24.9476,C -1.6724,E1 24.8909,E2 222.7775} C_DIS
LIN {X -74.6299,Y -75.5513,Z 110,A -139.1112,B 24.9467,C -1.6868,E1 24.8867,E2 224.8543} C_DIS
LIN {X -77.3061,Y -72.8106,Z 110,A -140.827,B 24.9456,C -1.7044,E1 24.8834,E2 226.5356} C_DIS
LIN {X -80.0733,Y -69.756,Z 110,A -143.3508,B 24.946,C -1.6982,E1 24.8787,E2 229.0854} C_DIS
LIN {X -82.298,Y -67.1175,Z 110,A -145.2073,B 24.9457,C -1.7028,E1 24.8754,E2 230.9396} C_DIS
LIN {X -84.7815,Y -63.9512,Z 110,A -147.3554,B 24.9453,C -1.7089,E1 24.8717,E2 233.0833} C_DIS
LIN {X -86.3924,Y -61.7574,Z 110,A -148.9224,B 24.9453,C -1.7089,E1 24.8691,E2 234.6579} C_DIS
LIN {X -88.3715,Y -58.8929,Z 110,A -150.8527,B 24.9451,C -1.7118,E1 24.8661,E2 236.5909} C_DIS
LIN {X -90.1026,Y -56.2062,Z 110,A -152.5577,B 24.9447,C -1.717,E1 24.8635,E2 238.2921} C_DIS
LIN {X -92.0551,Y -52.9478,Z 110,A -154.5991,B 24.9444,C -1.7228,E1 24.8606,E2 240.3304} C_DIS
LIN {X -93.836,Y -49.7242,Z 110,A -156.599,B 24.9441,C -1.7278,E1 24.858,E2 242.3289} C_DIS
LIN {X -95.3012,Y -46.8552,Z 110,A -158.3978,B 24.9439,C -1.7304,E1 24.8557,E2 244.1311} C_DIS
LIN {X -96.7675,Y -43.7456,Z 110,A -159.9914,B 24.9429,C -1.7452,E1 24.8539,E2 245.6981} C_DIS
LIN {X -99.1544,Y -38.0293,Z 110,A -163.6003,B 24.9429,C -1.7452,E1 24.85,E2 249.3272} C_DIS
LIN {X -100.599,Y -34.0216,Z 110,A -165.8778,B 24.9424,C -1.7528,E1 24.8479,E2 251.5995} C_DIS
LIN {X -101.608,Y -30.8832,Z 110,A -167.6583,B 24.9421,C -1.758,E1 24.8464,E2 253.3776} C_DIS
LIN {X -102.4907,Y -27.808,Z 110,A -169.3999,B 24.9418,C -1.7628,E1 24.8451,E2 255.118} C_DIS
LIN {X -103.3282,Y -24.5215,Z 110,A -171.416,B 24.9418,C -1.7617,E1 24.8438,E2 257.1485} C_DIS
LIN {X -104.176,Y -20.6225,Z 110,A -173.5247,B 24.9413,C -1.77,E1 24.8426,E2 259.2498} C_DIS
LIN {X -104.8617,Y -16.7916,Z 110,A -175.7714,B 24.9412,C -1.7714,E1 24.8415,E2 261.5067} C_DIS
LIN {X -105.4216,Y -12.8106,Z 110,A -177.8116,B 24.9404,C -1.7829,E1 24.8408,E2 263.5316} C_DIS
LIN {X -105.7972,Y -9.2126,Z 110,A -179.8842,B 24.9403,C -1.7848,E1 24.8403,E2 265.6121} C_DIS
LIN {X -106.0765,Y -5.0628,Z 110,A 177.965,B 24.9396,C -1.7953,E1 24.8399,E2 267.7507} C_DIS
LIN {X -106.1811,Y -1.7924,Z 110,A 176.2681,B 24.939,C -1.8035,E1 24.8398,E2 269.4383} C_DIS
LIN {X -106.1785,Y 1.9312,Z 110,A 174.4541,B 24.9381,C -1.817,E1 24.8398,E2 271.231} C_DIS
LIN {X -106.0649,Y 5.3061,Z 110,A 172.3194,B 24.9385,C -1.8117,E1 24.8401,E2 273.3914} C_DIS
LIN {X -105.7789,Y 9.4105,Z 110,A 170.1164,B 24.9379,C -1.8195,E1 24.8405,E2 275.5889} C_DIS
LIN {X -105.4069,Y 12.9363,Z 110,A 168.1578,B 24.9376,C -1.824,E1 24.8412,E2 277.5485} C_DIS
LIN {X -105.0493,Y 15.5778,Z 110,A 166.5551,B 24.9377,C -1.8228,E1 24.8418,E2 279.1636} C_DIS
LIN {X -104.3904,Y 19.5086,Z 110,A 164.5462,B 24.9369,C -1.8347,E1 24.8428,E2 281.1559} C_DIS
LIN {X -103.7214,Y 22.7928,Z 110,A 162.7748,B 24.9364,C -1.8419,E1 24.8438,E2 282.9207} C_DIS
LIN {X -102.8417,Y 26.4804,Z 110,A 160.756,B 24.9359,C -1.8493,E1 24.8452,E2 284.9335} C_DIS
LIN {X -102.0049,Y 29.5465,Z 110,A 159.0342,B 24.9355,C -1.8545,E1 24.8465,E2 286.653} C_DIS
LIN {X -100.9821,Y 32.8674,Z 110,A 157.0859,B 24.9353,C -1.8578,E1 24.8481,E2 288.6047} C_DIS
LIN {X -99.7635,Y 36.3986,Z 110,A 155.1141,B 24.9348,C -1.8656,E1 24.8499,E2 290.569} C_DIS
LIN {X -98.442,Y 39.8351,Z 110,A 153.0828,B 24.9344,C -1.8701,E1 24.852,E2 292.6008} C_DIS
LIN {X -97.3938,Y 42.3328,Z 110,A 151.6133,B 24.9341,C -1.8743,E1 24.8536,E2 294.0686} C_DIS
LIN {X -95.1867,Y 47.0861,Z 110,A 148.2607,B 24.9349,C -1.864,E1 24.8577,E2 297.4638} C_DIS
LIN {X -93.4701,Y 50.4086,Z 110,A 147.0283,B 24.9325,C -1.8982,E1 24.8592,E2 298.6215} C_DIS
LIN {X -91.1152,Y 54.5526,Z 110,A 144.0004,B 24.9331,C -1.8891,E1 24.8635,E2 301.6867} C_DIS
LIN {X -88.8924,Y 58.1028,Z 110,A 141.8097,B 24.9325,C -1.898,E1 24.8668,E2 303.8672} C_DIS
LIN {X -87.0131,Y 60.8806,Z 110,A 139.43,B 24.9336,C -1.8825,E1 24.8707,E2 306.2955} C_DIS
LIN {X -84.4997,Y 64.3257,Z 110,A 137.657,B 24.9318,C -1.9077,E1 24.8736,E2 308.017} C_DIS
LIN {X -81.7773,Y 67.7504,Z 110,A 135.3591,B 24.9312,C -1.9162,E1 24.8776,E2 310.3054} C_DIS
LIN {X -79.973,Y 69.8708,Z 110,A 132.9917,B 24.9331,C -1.8889,E1 24.8821,E2 312.7486} C_DIS
LIN {X -76.4846,Y 73.6731,Z 110,A 131.1418,B 24.9302,C -1.9295,E1 24.8855,E2 314.5097} C_DIS
LIN {X -74.0771,Y 76.0951,Z 110,A 129.2097,B 24.9302,C -1.9307,E1 24.8893,E2 316.4472} C_DIS
LIN {X -71.8393,Y 78.2095,Z 110,A 126.5646,B 24.9324,C -1.8989,E1 24.8949,E2 319.1786} C_DIS
LIN {X -67.6115,Y 81.8927,Z 110,A 124.2164,B 24.9302,C -1.9302,E1 24.8998,E2 321.4614} C_DIS
LIN {X -64.0176,Y 84.7316,Z 110,A 122.0112,B 24.9291,C -1.9452,E1 24.9046,E2 323.6389} C_DIS
LIN {X -60.7404,Y 87.1105,Z 110,A 119.8438,B 24.9287,C -1.9503,E1 24.9095,E2 325.8017} C_DIS
LIN {X -57.8746,Y 89.0422,Z 110,A 117.8657,B 24.9287,C -1.9497,E1 24.9142,E2 327.7877} C_DIS
LIN {X -55.4771,Y 90.5541,Z 110,A 116.1933,B 24.9289,C -1.9473,E1 24.9182,E2 329.4711} C_DIS
LIN {X -52.0544,Y 92.5638,Z 110,A 113.8777,B 24.9291,C -1.9446,E1 24.9238,E2 331.7998} C_DIS
LIN {X -49.2294,Y 94.0966,Z 110,A 112.5182,B 24.9279,C -1.9614,E1 24.9271,E2 333.123} C_DIS
LIN {X -45.8806,Y 95.7737,Z 110,A 110.5467,B 24.9275,C -1.9665,E1 24.932,E2 335.0877} C_DIS
LIN {X -42.8679,Y 97.1606,Z 110,A 108.5909,B 24.9278,C -1.963,E1 24.937,E2 337.0567} C_DIS
LIN {X -39.6318,Y 98.5248,Z 110,A 106.5675,B 24.9279,C -1.9608,E1 24.9423,E2 339.0897} C_DIS
LIN {X -35.5611,Y 100.066,Z 110,A 104.4295,B 24.9271,C -1.9718,E1 24.9478,E2 341.206} C_DIS
LIN {X -32.8195,Y 100.9976,Z 110,A 102.7126,B 24.9274,C -1.9678,E1 24.9524,E2 342.9354} C_DIS
LIN {X -29.1355,Y 102.1214,Z 110,A 100.8968,B 24.9265,C -1.98,E1 24.9572,E2 344.7252} C_DIS
LIN {X -26.419,Y 102.8574,Z 110,A 99.2538,B 24.9267,C -1.9769,E1 24.9616,E2 346.3783} C_DIS
LIN {X -21.8008,Y 103.9351,Z 110,A 96.4562,B 24.9272,C -1.9701,E1 24.9693,E2 349.1956} C_DIS
LIN {X -14.679,Y 105.177,Z 110,A 93.1081,B 24.9254,C -1.994,E1 24.9784,E2 352.4899} C_DIS
LIN {X -7.6139,Y 105.9238,Z 110,A 87.953,B 24.9291,C -1.9453,E1 24.9931,E2 357.7633} C_DIS
LIN {X -1.9048,Y 106.179,Z 110,A 85.9748,B 24.9259,C -1.9886,E1 24.9983,E2 359.6391} C_DIS
LIN {X 2.2525,Y 106.1717,Z 110,A 83.4977,B 24.9265,C -1.9799,E1 25.0053,E2 362.1366} C_DIS
LIN {X 6.8336,Y 105.9754,Z 110,A 80.7581,B 24.9273,C -1.9696,E1 25.013,E2 364.8995} C_DIS
LIN {X 10.208,Y 105.7053,Z 110,A 79.432,B 24.9258,C -1.9889,E1 25.0165,E2 366.179} C_DIS
LIN {X 14.1624,Y 105.2488,Z 110,A 77.0837,B 24.9265,C -1.9806,E1 25.0231,E2 368.5453} C_DIS
LIN {X 18.3599,Y 104.5979,Z 110,A 74.824,B 24.9265,C -1.9811,E1 25.0293,E2 370.8015} C_DIS
LIN {X 22.042,Y 103.8852,Z 110,A 72.7712,B 24.9265,C -1.979,E1 25.0349,E2 372.8567} C_DIS
LIN {X 26.2938,Y 102.8896,Z 110,A 70.514,B 24.9264,C -1.9816,E1 25.041,E2 375.1045} C_DIS
LIN {X 29.9577,Y 101.8833,Z 110,A 68.4261,B 24.9266,C -1.9787,E1 25.0466,E2 377.1959} C_DIS
LIN {X 33.516,Y 100.7695,Z 110,A 66.4511,B 24.9266,C -1.9785,E1 25.0519,E2 379.1676} C_DIS
LIN {X 36.6253,Y 99.6808,Z 110,A 64.5901,B 24.927,C -1.9736,E1 25.0568,E2 381.0364} C_DIS
LIN {X 39.9131,Y 98.4103,Z 110,A 62.4369,B 24.9279,C -1.9616,E1 25.0624,E2 383.2132} C_DIS
LIN {X 44.5204,Y 96.414,Z 110,A 60.0832,B 24.927,C -1.9727,E1 25.0684,E2 385.5346} C_DIS
LIN {X 47.2319,Y 95.1145,Z 110,A 58.5026,B 24.927,C -1.9724,E1 25.0723,E2 387.1118} C_DIS
LIN {X 50.4917,Y 93.425,Z 110,A 56.8286,B 24.9263,C -1.9823,E1 25.0764,E2 388.7578} C_DIS
LIN {X 52.8936,Y 92.0863,Z 110,A 54.9624,B 24.9276,C -1.9646,E1 25.081,E2 390.6603} C_DIS
LIN {X 55.3691,Y 90.6198,Z 110,A 53.3235,B 24.9281,C -1.9587,E1 25.085,E2 392.308} C_DIS
LIN {X 58.6637,Y 88.5225,Z 110,A 51.4186,B 24.9277,C -1.9636,E1 25.0894,E2 394.195} C_DIS
LIN {X 61.3731,Y 86.6666,Z 110,A 49.8307,B 24.9274,C -1.9682,E1 25.093,E2 395.7668} C_DIS
LIN {X 66.8479,Y 82.5165,Z 110,A 45.8241,B 24.9288,C -1.9491,E1 25.1019,E2 399.8038} C_DIS
LIN {X 69.9986,Y 79.8614,Z 110,A 43.6627,B 24.9289,C -1.9473,E1 25.1065,E2 401.961} C_DIS
LIN {X 72.7533,Y 77.36,Z 110,A 41.6843,B 24.9291,C -1.9444,E1 25.1106,E2 403.9383} C_DIS
LIN {X 75.4551,Y 74.7272,Z 110,A 38.7477,B 24.9321,C -1.9029,E1 25.1165,E2 406.9603} C_DIS
LIN {X 79.1824,Y 70.7656,Z 110,A 36.6886,B 24.93,C -1.9324,E1 25.1202,E2 408.9407} C_DIS
LIN {X 81.9719,Y 67.5162,Z 110,A 34.3689,B 24.9304,C -1.9266,E1 25.1244,E2 411.2636} C_DIS
LIN {X 84.2927,Y 64.5943,Z 110,A 32.3472,B 24.9308,C -1.9213,E1 25.1279,E2 413.2881} C_DIS
LIN {X 87.2446,Y 60.5475,Z 110,A 29.7741,B 24.9308,C -1.92,E1 25.132,E2 415.852} C_DIS
LIN {X 89.7219,Y 56.8157,Z 110,A 27.2357,B 24.9317,C -1.9085,E1 25.1359,E2 418.4046} C_DIS
LIN {X 91.6727,Y 53.6094,Z 110,A 25.2694,B 24.9319,C -1.9056,E1 25.1387,E2 420.3678} C_DIS
LIN {X 93.5775,Y 50.2105,Z 110,A 23.2299,B 24.9321,C -1.9025,E1 25.1415,E2 422.404} C_DIS
LIN {X 94.6803,Y 48.097,Z 110,A 21.4629,B 24.9338,C -1.8787,E1 25.1438,E2 424.2177} C_DIS
LIN {X 96.3235,Y 44.7147,Z 110,A 20.2854,B 24.9317,C -1.9088,E1 25.1451,E2 425.3178} C_DIS
LIN {X 97.7051,Y 41.6111,Z 110,A 18.0825,B 24.9332,C -1.8878,E1 25.1476,E2 427.5581} C_DIS
LIN {X 99.1095,Y 38.1478,Z 110,A 16.044,B 24.9337,C -1.8809,E1 25.1497,E2 429.6016} C_DIS
LIN {X 100.4598,Y 34.4343,Z 110,A 14.0005,B 24.9339,C -1.8783,E1 25.1516,E2 431.6398} C_DIS
LIN {X 101.4718,Y 31.3225,Z 110,A 12.0164,B 24.9349,C -1.8637,E1 25.1533,E2 433.6471} C_DIS
LIN {X 102.7037,Y 27.0172,Z 110,A 9.7766,B 24.9349,C -1.8637,E1 25.1549,E2 435.8739} C_DIS
LIN {X 103.5799,Y 23.4319,Z 110,A 7.9799,B 24.9347,C -1.8659,E1 25.1561,E2 437.6551} C_DIS
LIN {X 104.3993,Y 19.4625,Z 110,A 5.6755,B 24.9356,C -1.854,E1 25.1573,E2 439.9741} C_DIS
LIN {X 105.1571,Y 14.8188,Z 110,A 2.8795,B 24.9369,C -1.835,E1 25.1585,E2 442.7985} C_DIS
LIN {X 105.6226,Y 11.0218,Z 110,A 0.3686,B 24.9386,C -1.8095,E1 25.1593,E2 445.3548} C_DIS
LIN {X 106.0164,Y 6.1837,Z 110,A -1.6066,B 24.9373,C -1.8283,E1 25.1596,E2 447.2738} C_DIS
LIN {X 106.1924,Y 0.9836,Z 110,A -3.9559,B 24.9366,C -1.8389,E1 25.1598,E2 449.5842} C_DIS
LIN {X 106.0586,Y -5.4198,Z 110,A -7.773,B 24.9385,C -1.8121,E1 25.1595,E2 453.4418} C_DIS
LIN {X 105.7797,Y -9.4019,Z 110,A -9.9096,B 24.9389,C -1.8058,E1 25.159,E2 455.5805} C_DIS
LIN {X 105.37,Y -13.227,Z 110,A -12.3057,B 24.9403,C -1.7854,E1 25.1582,E2 458.0105} C_DIS
LIN {X 104.8906,Y -16.6051,Z 110,A -13.7957,B 24.9396,C -1.7944,E1 25.1576,E2 459.4705} C_DIS
LIN {X 104.2767,Y -20.0995,Z 110,A -15.6079,B 24.9398,C -1.7927,E1 25.1567,E2 461.2764} C_DIS
LIN {X 103.4905,Y -23.819,Z 110,A -17.6226,B 24.9401,C -1.7876,E1 25.1555,E2 463.2912} C_DIS
LIN {X 102.4481,Y -27.9655,Z 110,A -20.0291,B 24.9409,C -1.776,E1 25.1538,E2 465.7112} C_DIS
LIN {X 101.3948,Y -31.5708,Z 110,A -21.8503,B 24.9407,C -1.7784,E1 25.1523,E2 467.5165} C_DIS
LIN {X 100.2969,Y -34.903,Z 110,A -24.0151,B 24.9419,C -1.7608,E1 25.1504,E2 469.7106} C_DIS
LIN {X 98.5997,Y -39.4477,Z 110,A -26.4611,B 24.9419,C -1.76,E1 25.1479,E2 472.1449} C_DIS
LIN {X 97.1542,Y -42.8826,Z 110,A -28.8469,B 24.9434,C -1.7378,E1 25.1452,E2 474.5699} C_DIS
LIN {X 95.762,Y -45.9049,Z 110,A -30.232,B 24.9426,C -1.7499,E1 25.1436,E2 475.919} C_DIS
LIN {X 94.0712,Y -49.2776,Z 110,A -32.2478,B 24.943,C -1.7446,E1 25.141,E2 477.9365} C_DIS
LIN {X 92.551,Y -52.0773,Z 110,A -34.5439,B 24.9449,C -1.7151,E1 25.1378,E2 480.2904} C_DIS
LIN {X 90.415,Y -55.7059,Z 110,A -36.1747,B 24.9435,C -1.7357,E1 25.1355,E2 481.8643} C_DIS
LIN {X 88.8172,Y -58.2169,Z 110,A -37.7242,B 24.9437,C -1.7335,E1 25.1332,E2 483.4111} C_DIS
LIN {X 87.2117,Y -60.5948,Z 110,A -39.3391,B 24.9441,C -1.7263,E1 25.1306,E2 485.035} C_DIS
LIN {X 85.0476,Y -63.5969,Z 110,A -41.4491,B 24.9448,C -1.716,E1 25.1271,E2 487.1591} C_DIS
LIN {X 81.3657,Y -68.2456,Z 110,A -44.5927,B 24.9452,C -1.7099,E1 25.1216,E2 490.3027} C_DIS
LIN {X 79.0399,Y -70.9247,Z 110,A -46.3195,B 24.945,C -1.7129,E1 25.1184,E2 492.0147} C_DIS
LIN {X 76.0884,Y -74.0836,Z 110,A -49.1874,B 24.9468,C -1.6845,E1 25.1128,E2 494.9372} C_DIS
LIN {X 73.5923,Y -76.5625,Z 110,A -50.6361,B 24.9459,C -1.6988,E1 25.11,E2 496.3461} C_DIS
LIN {X 70.8437,Y -79.1125,Z 110,A -52.5926,B 24.946,C -1.6968,E1 25.106,E2 498.2993} C_DIS
LIN {X 67.5876,Y -81.9125,Z 110,A -55.0534,B 24.9468,C -1.6855,E1 25.1007,E2 500.7773} C_DIS
LIN {X 64.5979,Y -84.29,Z 110,A -57.0181,B 24.9468,C -1.685,E1 25.0964,E2 502.7357} C_DIS
LIN {X 61.6801,Y -86.4475,Z 110,A -58.8304,B 24.9467,C -1.687,E1 25.0923,E2 504.537} C_DIS
LIN {X 58.3829,Y -88.7077,Z 110,A -61.0611,B 24.9471,C -1.6796,E1 25.0871,E2 506.7777} C_DIS
LIN {X 55.7109,Y -90.412,Z 110,A -62.8496,B 24.9475,C -1.673,E1 25.0829,E2 508.5761} C_DIS
LIN {X 52.7,Y -92.1975,Z 110,A -64.5903,B 24.9474,C -1.6758,E1 25.0787,E2 510.305} C_DIS
LIN {X 49.8999,Y -93.7434,Z 110,A -66.4315,B 24.9479,C -1.6679,E1 25.0741,E2 512.1594} C_DIS
LIN {X 44.9208,Y -96.2276,Z 110,A -69.898,B 24.9494,C -1.644,E1 25.0653,E2 515.6734} C_DIS
LIN {X 41.4278,Y -97.7824,Z 110,A -71.9411,B 24.9494,C -1.6418,E1 25.06,E2 517.717} C_DIS
LIN {X 37.9213,Y -99.1953,Z 110,A -73.4122,B 24.9482,C -1.6622,E1 25.0564,E2 519.1365} C_DIS
LIN {X 34.943,Y -100.2829,Z 110,A -75.264,B 24.9487,C -1.6542,E1 25.0514,E2 521.0034} C_DIS
LIN {X 31.6224,Y -101.3789,Z 110,A -77.8628,B 24.9506,C -1.623,E1 25.0443,E2 523.6713} C_DIS
LIN {X 26.8107,Y -102.7567,Z 110,A -79.7467,B 24.9488,C -1.6532,E1 25.0395,E2 525.4808} C_DIS
LIN {X 23.5998,Y -103.5411,Z 110,A -81.5624,B 24.949,C -1.6501,E1 25.0345,E2 527.3012} C_DIS
LIN {X 19.9931,Y -104.2972,Z 110,A -83.4975,B 24.949,C -1.6506,E1 25.0292,E2 529.2328} C_DIS
LIN {X 13.6246,Y -105.3185,Z 110,A -86.9762,B 24.9491,C -1.6481,E1 25.0196,E2 532.7141} C_DIS
LIN {X 9.9235,Y -105.7316,Z 110,A -88.9996,B 24.9492,C -1.6464,E1 25.014,E2 534.7403} C_DIS
LIN {X 6.1926,Y -106.0159,Z 110,A -91.0704,B 24.9494,C -1.6434,E1 25.0082,E2 536.8172} C_DIS
LIN {X 2.5481,Y -106.1672,Z 110,A -92.9469,B 24.9492,C -1.6464,E1 25.003,E2 538.6863} C_DIS
LIN {X 2.5481,Y -106.1672,Z 110,A -92.9469,B 24.9492,C -1.6464,E1 25.003,E2 538.6863} C_DIS
Enddeposition()
LIN {X 0.7467,Y -105.2494,Z 110,A -93.6132,B 24.9474,C -1.6749,E1 25.0013,E2 539.2848} C_DIS
Startdeposition()
$VEL.CP = VEL_PRINT
LIN {X 3.0455,Y -105.2081,Z 110,A -91.9256,B 24.9463,C -1.6927,E1 25.0061,E2 537.5553} C_DIS
LIN {X 6.4495,Y -105.0562,Z 110,A -90.1387,B 24.9464,C -1.6907,E1 25.0111,E2 535.7739} C_DIS
LIN {X 9.482,Y -104.8242,Z 110,A -88.402,B 24.9462,C -1.6948,E1 25.016,E2 534.0283} C_DIS
LIN {X 12.8836,Y -104.4625,Z 110,A -86.6248,B 24.9463,C -1.6924,E1 25.0209,E2 532.258} C_DIS
LIN {X 15.478,Y -104.1095,Z 110,A -85.2054,B 24.9463,C -1.6932,E1 25.0248,E2 530.838} C_DIS
LIN {X 18.4682,Y -103.6192,Z 110,A -83.4682,B 24.946,C -1.6981,E1 25.0296,E2 529.0911} C_DIS
LIN {X 21.347,Y -103.0647,Z 110,A -81.9021,B 24.946,C -1.6982,E1 25.0339,E2 527.5265} C_DIS
LIN {X 24.756,Y -102.2994,Z 110,A -79.9738,B 24.9458,C -1.7011,E1 25.0391,E2 525.594} C_DIS
LIN {X 28.0397,Y -101.4502,Z 110,A -78.064,B 24.9455,C -1.7057,E1 25.0443,E2 523.6765} C_DIS
LIN {X 31.2854,Y -100.4949,Z 110,A -76.3732,B 24.9457,C -1.7016,E1 25.0488,E2 521.9983} C_DIS
LIN {X 34.2338,Y -99.5311,Z 110,A -74.7002,B 24.9457,C -1.7031,E1 25.0532,E2 520.3251} C_DIS
LIN {X 36.2262,Y -98.8214,Z 110,A -73.4902,B 24.9454,C -1.707,E1 25.0564,E2 519.1082} C_DIS
LIN {X 39.5268,Y -97.5482,Z 110,A -71.547,B 24.9452,C -1.7105,E1 25.0615,E2 517.1612} C_DIS
LIN {X 42.215,Y -96.4153,Z 110,A -70.0654,B 24.9453,C -1.7084,E1 25.0653,E2 515.6881} C_DIS
LIN {X 44.959,Y -95.1685,Z 110,A -68.2643,B 24.9447,C -1.7176,E1 25.0699,E2 513.8697} C_DIS
LIN {X 47.9642,Y -93.688,Z 110,A -66.5768,B 24.9449,C -1.715,E1 25.074,E2 512.193} C_DIS
LIN {X 50.7381,Y -92.2173,Z 110,A -64.8981,B 24.9448,C -1.7167,E1 25.0782,E2 510.5151} C_DIS
LIN {X 52.9976,Y -90.9377,Z 110,A -63.4861,B 24.9446,C -1.7192,E1 25.0816,E2 509.1014} C_DIS
LIN {X 55.2091,Y -89.6122,Z 110,A -62.0899,B 24.9445,C -1.7215,E1 25.0849,E2 507.7041} C_DIS
LIN {X 57.363,Y -88.2487,Z 110,A -60.3786,B 24.9434,C -1.7378,E1 25.089,E2 505.9599} C_DIS
LIN {X 61.2799,Y -85.5734,Z 110,A -58.0751,B 24.9438,C -1.7314,E1 25.0942,E2 503.6795} C_DIS
LIN {X 63.7246,Y -83.771,Z 110,A -56.397,B 24.9435,C -1.7359,E1 25.098,E2 501.9967} C_DIS
LIN {X 66.2573,Y -81.78,Z 110,A -54.6953,B 24.9435,C -1.7376,E1 25.1017,E2 500.2974} C_DIS
LIN {X 68.7569,Y -79.6924,Z 110,A -52.8284,B 24.9429,C -1.7456,E1 25.1057,E2 498.419} C_DIS
LIN {X 71.1563,Y -77.555,Z 110,A -51.1917,B 24.9429,C -1.745,E1 25.1091,E2 496.7903} C_DIS
LIN {X 73.4894,Y -75.3504,Z 110,A -49.3541,B 24.9424,C -1.753,E1 25.1128,E2 494.9414} C_DIS
LIN {X 75.7555,Y -73.0692,Z 110,A -47.6707,B 24.9424,C -1.7545,E1 25.1161,E2 493.2616} C_DIS
LIN {X 78.2647,Y -70.3752,Z 110,A -45.7021,B 24.9421,C -1.7581,E1 25.1198,E2 491.2933} C_DIS
LIN {X 80.2605,Y -68.0904,Z 110,A -44.0742,B 24.9419,C -1.7614,E1 25.1228,E2 489.665} C_DIS
LIN {X 82.4135,Y -65.4681,Z 110,A -42.2211,B 24.9415,C -1.7665,E1 25.126,E2 487.8082} C_DIS
LIN {X 84.2661,Y -63.0655,Z 110,A -40.6466,B 24.9415,C -1.7678,E1 25.1287,E2 486.2384} C_DIS
LIN {X 85.7364,Y -61.0513,Z 110,A -39.2167,B 24.941,C -1.7746,E1 25.131,E2 484.7993} C_DIS
LIN {X 87.2502,Y -58.8679,Z 110,A -37.7976,B 24.9408,C -1.7775,E1 25.1332,E2 483.3804} C_DIS
LIN {X 89.1628,Y -55.9288,Z 110,A -35.8804,B 24.9404,C -1.7833,E1 25.1361,E2 481.4591} C_DIS
LIN {X 90.6436,Y -53.4951,Z 110,A -34.4368,B 24.9404,C -1.7832,E1 25.1382,E2 480.0232} C_DIS
LIN {X 91.9389,Y -51.2371,Z 110,A -32.9948,B 24.9401,C -1.7884,E1 25.1402,E2 478.5764} C_DIS
LIN {X 93.4301,Y -48.4687,Z 110,A -31.3131,B 24.9398,C -1.7922,E1 25.1424,E2 476.8946} C_DIS
LIN {X 94.5882,Y -46.1679,Z 110,A -29.7426,B 24.939,C -1.8036,E1 25.1443,E2 475.3055} C_DIS
LIN {X 96.0394,Y -43.0634,Z 110,A -28.0065,B 24.939,C -1.8038,E1 25.1463,E2 473.5786} C_DIS
LIN {X 97.2395,Y -40.285,Z 110,A -26.4301,B 24.9389,C -1.8057,E1 25.1481,E2 472.0061} C_DIS
LIN {X 98.1922,Y -37.9033,Z 110,A -24.8825,B 24.9381,C -1.8166,E1 25.1497,E2 470.4415} C_DIS
LIN {X 99.357,Y -34.7302,Z 110,A -23.2164,B 24.9383,C -1.8149,E1 25.1512,E2 468.7888} C_DIS
LIN {X 100.2293,Y -32.1272,Z 110,A -21.6909,B 24.9379,C -1.8209,E1 25.1525,E2 467.2577} C_DIS
LIN {X 100.956,Y -29.764,Z 110,A -20.3316,B 24.9375,C -1.8257,E1 25.1536,E2 465.8948} C_DIS
LIN {X 101.8977,Y -26.3603,Z 110,A -18.3963,B 24.9371,C -1.8324,E1 25.155,E2 463.9547} C_DIS
LIN {X 102.5931,Y -23.5091,Z 110,A -16.8371,B 24.9368,C -1.8359,E1 25.156,E2 462.3964} C_DIS
LIN {X 103.3176,Y -20.0873,Z 110,A -14.916,B 24.9363,C -1.8427,E1 25.1571,E2 460.4704} C_DIS
LIN {X 103.9136,Y -16.7434,Z 110,A -13.1692,B 24.9363,C -1.8443,E1 25.1579,E2 458.7302} C_DIS
LIN {X 104.351,Y -13.7443,Z 110,A -11.4306,B 24.9356,C -1.8535,E1 25.1586,E2 456.9801} C_DIS
LIN {X 104.748,Y -10.3077,Z 110,A -9.6651,B 24.9356,C -1.8545,E1 25.1591,E2 455.2227} C_DIS
LIN {X 104.9691,Y -7.7388,Z 110,A -8.2687,B 24.9352,C -1.8587,E1 25.1594,E2 453.8246} C_DIS
LIN {X 105.1329,Y -5.0325,Z 110,A -6.4999,B 24.934,C -1.8762,E1 25.1597,E2 452.0251} C_DIS
LIN {X 105.2516,Y -0.5032,Z 110,A -4.3238,B 24.9343,C -1.8717,E1 25.1597,E2 449.8727} C_DIS
LIN {X 105.2231,Y 2.5408,Z 110,A -2.7066,B 24.9341,C -1.8753,E1 25.1597,E2 448.2566} C_DIS
LIN {X 105.1323,Y 5.0461,Z 110,A -1.1487,B 24.9332,C -1.888,E1 25.1595,E2 446.6779} C_DIS
LIN {X 104.907,Y 8.5168,Z 110,A 0.5769,B 24.9332,C -1.8869,E1 25.1592,E2 444.9651} C_DIS
LIN {X 104.5716,Y 11.9526,Z 110,A 2.5074,B 24.9327,C -1.8951,E1 25.1586,E2 443.0267} C_DIS
LIN {X 104.1331,Y 15.3154,Z 110,A 4.225,B 24.9327,C -1.8954,E1 25.1579,E2 441.3184} C_DIS
LIN {X 103.623,Y 18.4472,Z 110,A 6.0331,B 24.932,C -1.9044,E1 25.1571,E2 439.4999} C_DIS
LIN {X 103.0697,Y 21.3227,Z 110,A 7.5947,B 24.9318,C -1.908,E1 25.1562,E2 437.9389} C_DIS
LIN {X 102.4063,Y 24.3177,Z 110,A 9.1869,B 24.9316,C -1.9098,E1 25.1552,E2 436.3516} C_DIS
LIN {X 101.5656,Y 27.6123,Z 110,A 11.0248,B 24.9313,C -1.915,E1 25.1539,E2 434.5121} C_DIS
LIN {X 100.7283,Y 30.5316,Z 110,A 12.6623,B 24.9309,C -1.9193,E1 25.1526,E2 432.8737} C_DIS
LIN {X 99.5298,Y 34.2377,Z 110,A 14.7746,B 24.9305,C -1.9254,E1 25.1508,E2 430.7591} C_DIS
LIN {X 98.82,Y 36.2302,Z 110,A 15.9802,B 24.9301,C -1.9311,E1 25.1496,E2 429.5466} C_DIS
LIN {X 97.541,Y 39.5444,Z 110,A 17.9203,B 24.9297,C -1.9371,E1 25.1476,E2 427.6033} C_DIS
LIN {X 96.2185,Y 42.666,Z 110,A 19.8439,B 24.929,C -1.9457,E1 25.1455,E2 425.6699} C_DIS
LIN {X 94.7974,Y 45.7326,Z 110,A 21.5643,B 24.929,C -1.9459,E1 25.1434,E2 423.9583} C_DIS
LIN {X 93.0425,Y 49.2049,Z 110,A 23.6688,B 24.9286,C -1.9512,E1 25.1408,E2 421.8524} C_DIS
LIN {X 91.8099,Y 51.4681,Z 110,A 25.0642,B 24.9284,C -1.9547,E1 25.1389,E2 420.4559} C_DIS
LIN {X 89.9967,Y 54.5764,Z 110,A 27.0171,B 24.928,C -1.9597,E1 25.1361,E2 418.5013} C_DIS
LIN {X 88.4781,Y 57.0058,Z 110,A 28.5645,B 24.9277,C -1.9633,E1 25.1338,E2 416.9533} C_DIS
LIN {X 86.7933,Y 59.5426,Z 110,A 30.1493,B 24.9277,C -1.9644,E1 25.1313,E2 415.3736} C_DIS
LIN {X 84.541,Y 62.6995,Z 110,A 32.3465,B 24.927,C -1.9733,E1 25.1277,E2 413.166} C_DIS
LIN {X 82.5789,Y 65.2589,Z 110,A 34.0739,B 24.9268,C -1.9764,E1 25.1247,E2 411.4394} C_DIS
LIN {X 80.2757,Y 68.0725,Z 110,A 36.0328,B 24.9265,C -1.9802,E1 25.1212,E2 409.4805} C_DIS
LIN {X 78.295,Y 70.3414,Z 110,A 37.7057,B 24.9261,C -1.9854,E1 25.1181,E2 407.8029} C_DIS
LIN {X 75.7664,Y 73.0578,Z 110,A 39.702,B 24.9258,C -1.9889,E1 25.1143,E2 405.8071} C_DIS
LIN {X 73.2095,Y 75.6202,Z 110,A 41.6352,B 24.9256,C -1.9915,E1 25.1104,E2 403.8758} C_DIS
LIN {X 70.8599,Y 77.8269,Z 110,A 43.4895,B 24.9251,C -1.9992,E1 25.1066,E2 402.0109} C_DIS
LIN {X 68.2224,Y 80.148,Z 110,A 45.3115,B 24.9251,C -1.9992,E1 25.1028,E2 400.1959} C_DIS
LIN {X 65.3213,Y 82.5295,Z 110,A 47.3295,B 24.9248,C -2.002,E1 25.0984,E2 398.1789} C_DIS
LIN {X 62.4097,Y 84.7532,Z 110,A 49.436,B 24.9242,C -2.0102,E1 25.0937,E2 396.0607} C_DIS
LIN {X 59.551,Y 86.7875,Z 110,A 51.144,B 24.9246,C -2.0051,E1 25.0898,E2 394.3707} C_DIS
LIN {X 57.4006,Y 88.2246,Z 110,A 52.7144,B 24.9239,C -2.014,E1 25.0861,E2 392.7843} C_DIS
LIN {X 54.5294,Y 90.0253,Z 110,A 54.4539,B 24.9241,C -2.0125,E1 25.082,E2 391.0538} C_DIS
LIN {X 51.4022,Y 91.8467,Z 110,A 56.4189,B 24.9239,C -2.0152,E1 25.0772,E2 389.0885} C_DIS
LIN {X 48.4715,Y 93.4287,Z 110,A 58.1584,B 24.9239,C -2.0146,E1 25.0729,E2 387.3553} C_DIS
LIN {X 46.5844,Y 94.3818,Z 110,A 59.3679,B 24.9236,C -2.0184,E1 25.0699,E2 386.1399} C_DIS
LIN {X 43.84,Y 95.6893,Z 110,A 60.9551,B 24.9236,C -2.0176,E1 25.0659,E2 384.5587} C_DIS
LIN {X 41.4796,Y 96.7359,Z 110,A 62.3575,B 24.9236,C -2.0191,E1 25.0623,E2 383.1563} C_DIS
LIN {X 39.115,Y 97.7158,Z 110,A 63.9199,B 24.9229,C -2.0273,E1 25.0582,E2 381.5779} C_DIS
LIN {X 36.0351,Y 98.8912,Z 110,A 65.5736,B 24.9232,C -2.0234,E1 25.0539,E2 379.9371} C_DIS
LIN {X 33.4536,Y 99.7942,Z 110,A 67.0874,B 24.9231,C -2.0257,E1 25.0499,E2 378.4209} C_DIS
LIN {X 30.5565,Y 100.7209,Z 110,A 68.6793,B 24.9231,C -2.0244,E1 25.0457,E2 376.8349} C_DIS
LIN {X 28.0795,Y 101.4393,Z 110,A 70.2496,B 24.9226,C -2.032,E1 25.0414,E2 375.2491} C_DIS
LIN {X 24.7844,Y 102.2925,Z 110,A 71.936,B 24.923,C -2.0265,E1 25.0369,E2 373.5783} C_DIS
LIN {X 22.252,Y 102.8731,Z 110,A 73.4059,B 24.9228,C -2.0294,E1 25.0329,E2 372.1035} C_DIS
LIN {X 19.2735,Y 103.4743,Z 110,A 75.1646,B 24.9224,C -2.0342,E1 25.028,E2 370.3353} C_DIS
LIN {X 15.921,Y 104.041,Z 110,A 76.8497,B 24.9229,C -2.0283,E1 25.0234,E2 368.666} C_DIS
LIN {X 12.9005,Y 104.4603,Z 110,A 78.6826,B 24.9223,C -2.0354,E1 25.0183,E2 366.8176} C_DIS
LIN {X 9.4973,Y 104.8228,Z 110,A 80.4287,B 24.9226,C -2.0311,E1 25.0135,E2 365.083} C_DIS
LIN {X 6.5041,Y 105.0526,Z 110,A 82.1504,B 24.9224,C -2.0345,E1 25.0087,E2 363.3539} C_DIS
LIN {X 3.1818,Y 105.2039,Z 110,A 83.7997,B 24.9229,C -2.0281,E1 25.0041,E2 361.7201} C_DIS
LIN {X 0.3185,Y 105.2521,Z 110,A 85.4051,B 24.9228,C -2.0297,E1 24.9996,E2 360.1112} C_DIS
LIN {X -3.0284,Y 105.2086,Z 110,A 87.286,B 24.9226,C -2.0315,E1 24.9944,E2 358.2259} C_DIS
LIN {X -6.3961,Y 105.0592,Z 110,A 89.033,B 24.9229,C -2.0274,E1 24.9895,E2 356.4881} C_DIS
LIN {X -9.4672,Y 104.8256,Z 110,A 90.8001,B 24.9227,C -2.0301,E1 24.9846,E2 354.7137} C_DIS
LIN {X -12.8017,Y 104.4721,Z 110,A 92.5223,B 24.9231,C -2.0251,E1 24.9798,E2 353.0024} C_DIS
LIN {X -15.2415,Y 104.1436,Z 110,A 93.8936,B 24.9231,C -2.0255,E1 24.976,E2 351.6291} C_DIS
LIN {X -18.3942,Y 103.6325,Z 110,A 95.7139,B 24.9229,C -2.0273,E1 24.971,E2 349.8026} C_DIS
LIN {X -21.2276,Y 103.0892,Z 110,A 97.2663,B 24.9231,C -2.0253,E1 24.9667,E2 348.2532} C_DIS
LIN {X -24.2748,Y 102.4162,Z 110,A 98.8993,B 24.9234,C -2.0213,E1 24.9623,E2 346.6278} C_DIS
LIN {X -26.3706,Y 101.8951,Z 110,A 100.1382,B 24.9233,C -2.0225,E1 24.959,E2 345.384} C_DIS
LIN {X -29.7449,Y 100.9617,Z 110,A 102.0784,B 24.9233,C -2.0218,E1 24.9537,E2 343.4424} C_DIS
LIN {X -32.55,Y 100.0925,Z 110,A 103.6084,B 24.9237,C -2.0173,E1 24.9497,E2 341.9204} C_DIS
LIN {X -35.4568,Y 99.1021,Z 110,A 105.2652,B 24.9239,C -2.0146,E1 24.9453,E2 340.2667} C_DIS
LIN {X -37.8406,Y 98.2163,Z 110,A 106.8304,B 24.9235,C -2.0196,E1 24.9412,E2 338.6863} C_DIS
LIN {X -41.0482,Y 96.9178,Z 110,A 108.5433,B 24.9242,C -2.0106,E1 24.9368,E2 336.9912} C_DIS
LIN {X -43.5301,Y 95.8291,Z 110,A 110.0042,B 24.9244,C -2.0078,E1 24.9331,E2 335.5333} C_DIS
LIN {X -45.7389,Y 94.7944,Z 110,A 111.4186,B 24.9244,C -2.009,E1 24.9295,E2 334.1125} C_DIS
LIN {X -48.4552,Y 93.437,Z 110,A 113.1793,B 24.9242,C -2.0103,E1 24.9251,E2 332.344} C_DIS
LIN {X -51.4432,Y 91.8238,Z 110,A 114.9412,B 24.9247,C -2.0039,E1 24.9209,E2 330.5923} C_DIS
LIN {X -54.5223,Y 90.0296,Z 110,A 116.9065,B 24.9249,C -2.0013,E1 24.9161,E2 328.6272} C_DIS
LIN {X -57.0108,Y 88.4748,Z 110,A 118.4828,B 24.9252,C -1.9975,E1 24.9124,E2 327.0549} C_DIS
LIN {X -59.9228,Y 86.5291,Z 110,A 120.4265,B 24.9254,C -1.9951,E1 24.9079,E2 325.1104} C_DIS
LIN {X -62.3196,Y 84.8192,Z 110,A 122.0104,B 24.9257,C -1.9911,E1 24.9044,E2 323.5304} C_DIS
LIN {X -64.5681,Y 83.1211,Z 110,A 123.6106,B 24.9257,C -1.9902,E1 24.9008,E2 321.9264} C_DIS
LIN {X -67.2667,Y 80.9517,Z 110,A 125.429,B 24.9262,C -1.9837,E1 24.8969,E2 320.1168} C_DIS
LIN {X -69.6896,Y 78.8778,Z 110,A 127.3313,B 24.9261,C -1.9858,E1 24.8929,E2 318.2019} C_DIS
LIN {X -72.2737,Y 76.515,Z 110,A 129.0932,B 24.9268,C -1.9761,E1 24.8893,E2 316.4561} C_DIS
LIN {X -74.7101,Y 74.138,Z 110,A 130.9731,B 24.927,C -1.9726,E1 24.8856,E2 314.5765} C_DIS
LIN {X -76.9237,Y 71.8391,Z 110,A 132.8051,B 24.9271,C -1.9717,E1 24.882,E2 312.7386} C_DIS
LIN {X -79.2743,Y 69.2356,Z 110,A 134.6215,B 24.9277,C -1.9635,E1 24.8787,E2 310.9337} C_DIS
LIN {X -81.3579,Y 66.7779,Z 110,A 136.4954,B 24.9277,C -1.9632,E1 24.8753,E2 309.0517} C_DIS
LIN {X -83.368,Y 64.2477,Z 110,A 138.144,B 24.9284,C -1.9545,E1 24.8725,E2 307.4161} C_DIS
LIN {X -85.2853,Y 61.6829,Z 110,A 140.0559,B 24.9283,C -1.9559,E1 24.8694,E2 305.4917} C_DIS
LIN {X -87.2534,Y 58.8631,Z 110,A 141.745,B 24.9291,C -1.9441,E1 24.8667,E2 303.8223} C_DIS
LIN {X -88.9253,Y 56.3089,Z 110,A 143.4143,B 24.9295,C -1.9396,E1 24.8642,E2 302.1553} C_DIS
LIN {X -90.0361,Y 54.5116,Z 110,A 144.6341,B 24.9295,C -1.9389,E1 24.8624,E2 300.931} C_DIS
LIN {X -91.814,Y 51.4607,Z 110,A 146.5924,B 24.9298,C -1.9346,E1 24.8597,E2 298.9726} C_DIS
LIN {X -93.4148,Y 48.4979,Z 110,A 148.3519,B 24.9304,C -1.9265,E1 24.8574,E2 297.2231} C_DIS
LIN {X -94.5598,Y 46.2251,Z 110,A 149.8885,B 24.9304,C -1.9278,E1 24.8555,E2 295.675} C_DIS
LIN {X -95.9662,Y 43.2259,Z 110,A 151.6484,B 24.9308,C -1.9209,E1 24.8534,E2 293.9223} C_DIS
LIN {X -97.2414,Y 40.2805,Z 110,A 153.3202,B 24.9314,C -1.9128,E1 24.8516,E2 292.2605} C_DIS
LIN {X -98.1985,Y 37.8873,Z 110,A 154.9016,B 24.9313,C -1.9149,E1 24.85,E2 290.6651} C_DIS
LIN {X -99.3701,Y 34.693,Z 110,A 156.6611,B 24.9319,C -1.9058,E1 24.8484,E2 288.9174} C_DIS
LIN {X -100.4816,Y 31.3283,Z 110,A 158.6289,B 24.9322,C -1.9011,E1 24.8467,E2 286.9494} C_DIS
LIN {X -101.4436,Y 28.0641,Z 110,A 160.4045,B 24.9329,C -1.8925,E1 24.8453,E2 285.1842} C_DIS
LIN {X -102.1006,Y 25.5708,Z 110,A 161.8172,B 24.9332,C -1.8883,E1 24.8444,E2 283.773} C_DIS
LIN {X -102.8727,Y 22.2536,Z 110,A 163.7474,B 24.9334,C -1.8852,E1 24.8432,E2 281.8391} C_DIS
LIN {X -103.4743,Y 19.2734,Z 110,A 165.3507,B 24.9339,C -1.878,E1 24.8423,E2 280.2435} C_DIS
Enddeposition()
END
